LIN {X 0,Y 502.137,Z 842.26,A -85,B 0,C 180,E1 13995.84,E2 13995.84} C_VEL
LIN {X 0,Y 481.443,Z 805.869,A -85,B 0,C 180,E1 13999.134,E2 13999.134} C_VEL
LIN {X 0,Y 469.956,Z 788.258,A -85,B 0,C 180,E1 14001.102,E2 14001.102} C_VEL
LIN {X 0,Y 468.202,Z 783.31,A -85,B 0,C 180,E1 14001.543,E2 14001.543} C_VEL
LIN {X 0,Y 468.344,Z 783.31,A -85,B 0,C 180,E1 14007.257,E2 14007.257} C_VEL
LIN {X 0,Y 468.598,Z 783.31,A -85,B 0,C 180,E1 14013.095,E2 14013.095} C_VEL
LIN {X 0,Y 468.809,Z 783.31,A -85,B 0,C 180,E1 14019.592,E2 14019.592} C_VEL
LIN {X 0,Y 468.958,Z 783.31,A -85,B 0,C 180,E1 14025.753,E2 14025.753} C_VEL
LIN {X 0,Y 469.248,Z 783.31,A -85,B 0,C 180,E1 14030.717,E2 14030.717} C_VEL
LIN {X 0,Y 469.562,Z 783.31,A -85,B 0,C 180,E1 14036.307,E2 14036.307} C_VEL
LIN {X 0,Y 469.678,Z 783.31,A -85,B 0,C 180,E1 14041.855,E2 14041.855} C_VEL
LIN {X 0,Y 469.329,Z 783.31,A -85,B 0,C 180,E1 14047.426,E2 14047.426} C_VEL
LIN {X 0,Y 469.059,Z 783.31,A -85,B 0,C 180,E1 14053.074,E2 14053.074} C_VEL
LIN {X 0,Y 468.787,Z 783.31,A -85,B 0,C 180,E1 14058.863,E2 14058.863} C_VEL
LIN {X 0,Y 468.495,Z 783.31,A -85,B 0,C 180,E1 14065.107,E2 14065.107} C_VEL
LIN {X 0,Y 468.32,Z 783.31,A -85,B 0,C 180,E1 14071.18,E2 14071.18} C_VEL
LIN {X 0,Y 468.157,Z 783.31,A -85,B 0,C 180,E1 14077.951,E2 14077.951} C_VEL
LIN {X 0,Y 468.177,Z 783.696,A -85,B 0,C 180,E1 14081.783,E2 14081.783} C_VEL
LIN {X 0,Y 470.703,Z 789.093,A -85,B 0,C 180,E1 14082.265,E2 14082.265} C_VEL
LIN {X 0,Y 493.353,Z 825.509,A -85,B 0,C 180,E1 14085.963,E2 14085.963} C_VEL
LIN {X 0,Y 512.919,Z 863.779,A -85,B 0,C 180,E1 14089.04,E2 14089.04} C_VEL
LIN {X 0,Y 517.833,Z 877.244,A -85,B 0,C 180,E1 14089.994,E2 14089.994} C_VEL
LIN {X 0,Y 512.74,Z 919.111,A -85,B 0,C 180,E1 14091.466,E2 14091.466} C_VEL
LIN {X 0,Y 506.507,Z 957.08,A -85,B 0,C 180,E1 14093.46,E2 14093.46} C_VEL
LIN {X 0,Y 499.069,Z 993.486,A -85,B 0,C 180,E1 14096.094,E2 14096.094} C_VEL
LIN {X 0,Y 490.992,Z 1028.436,A -85,B 0,C 180,E1 14099.537,E2 14099.537} C_VEL
LIN {X 0,Y 483.283,Z 1059.873,A -85,B 0,C 180,E1 14103.731,E2 14103.731} C_VEL
LIN {X 0,Y 477.35,Z 1085.407,A -85,B 0,C 180,E1 14108.348,E2 14108.348} C_VEL
LIN {X 0,Y 473.318,Z 1105.246,A -85,B 0,C 180,E1 14113.257,E2 14113.257} C_VEL
LIN {X 0,Y 471.002,Z 1119.649,A -85,B 0,C 180,E1 14118.403,E2 14118.403} C_VEL
LIN {X 0,Y 470.112,Z 1128.462,A -85,B 0,C 180,E1 14123.525,E2 14123.525} C_VEL
LIN {X 0,Y 469.91,Z 1132.17,A -85,B 0,C 180,E1 14128.344,E2 14128.344} C_VEL
LIN {X 0,Y 469.969,Z 1131.123,A -85,B 0,C 180,E1 14133.699,E2 14133.699} C_VEL
LIN {X 0,Y 470.403,Z 1125.694,A -85,B 0,C 180,E1 14138.336,E2 14138.336} C_VEL
LIN {X 0,Y 471.702,Z 1114.802,A -85,B 0,C 180,E1 14143.468,E2 14143.468} C_VEL
LIN {X 0,Y 474.604,Z 1098.044,A -85,B 0,C 180,E1 14148.619,E2 14148.619} C_VEL
LIN {X 0,Y 479.46,Z 1075.81,A -85,B 0,C 180,E1 14153.465,E2 14153.465} C_VEL
LIN {X 0,Y 486.177,Z 1048.272,A -85,B 0,C 180,E1 14157.872,E2 14157.872} C_VEL
LIN {X 0,Y 493.802,Z 1016.531,A -85,B 0,C 180,E1 14161.662,E2 14161.662} C_VEL
LIN {X 0,Y 502.224,Z 978.76,A -85,B 0,C 180,E1 14164.976,E2 14164.976} C_VEL
LIN {X 0,Y 509.443,Z 940.342,A -85,B 0,C 180,E1 14167.412,E2 14167.412} C_VEL
LIN {X 0,Y 515.66,Z 896.96,A -85,B 0,C 180,E1 14169.309,E2 14169.309} C_VEL
LIN {X 0,Y 517.573,Z 874.805,A -85,B 0,C 180,E1 14170.015,E2 14170.015} C_VEL
LIN {X 0,Y 499.743,Z 836.77,A -85,B 0,C 180,E1 14172.967,E2 14172.967} C_VEL
LIN {X 0,Y 477.929,Z 800.29,A -85,B 0,C 180,E1 14176.384,E2 14176.384} C_VEL
LIN {X 0,Y 468.27,Z 784.748,A -85,B 0,C 180,E1 14178.066,E2 14178.066} C_VEL
LIN {X 0,Y 468.127,Z 783.31,A -85,B 0,C 180,E1 14178.331,E2 14178.331} C_VEL
LIN {X 0,Y 468.144,Z 783.31,A -85,B 0,C 180,E1 14184.363,E2 14184.363} C_VEL
LIN {X 0,Y 468.406,Z 783.31,A -85,B 0,C 180,E1 14190.856,E2 14190.856} C_VEL
LIN {X 0,Y 468.695,Z 783.31,A -85,B 0,C 180,E1 14197.169,E2 14197.169} C_VEL
LIN {X 0,Y 468.892,Z 783.31,A -85,B 0,C 180,E1 14203.087,E2 14203.087} C_VEL
LIN {X 0,Y 469.159,Z 783.31,A -85,B 0,C 180,E1 14208.821,E2 14208.821} C_VEL
LIN {X 0,Y 469.481,Z 783.31,A -85,B 0,C 180,E1 14214.438,E2 14214.438} C_VEL
LIN {X 0,Y 469.716,Z 783.31,A -85,B 0,C 180,E1 14220.197,E2 14220.197} C_VEL
LIN {X 0,Y 469.484,Z 783.31,A -85,B 0,C 180,E1 14225.549,E2 14225.549} C_VEL
LIN {X 0,Y 469.164,Z 783.31,A -85,B 0,C 180,E1 14231.165,E2 14231.165} C_VEL
LIN {X 0,Y 468.934,Z 783.31,A -85,B 0,C 180,E1 14236.897,E2 14236.897} C_VEL
LIN {X 0,Y 468.69,Z 783.31,A -85,B 0,C 180,E1 14242.816,E2 14242.816} C_VEL
LIN {X 0,Y 468.44,Z 783.31,A -85,B 0,C 180,E1 14249.151,E2 14249.151} C_VEL
LIN {X 0,Y 468.192,Z 783.31,A -85,B 0,C 180,E1 14255.615,E2 14255.615} C_VEL
LIN {X 0,Y 468.162,Z 783.31,A -85,B 0,C 180,E1 14258.52,E2 14258.52} C_VEL
LIN {X 0,Y 470.442,Z 788.792,A -85,B 0,C 180,E1 14259.003,E2 14259.003} C_VEL
LIN {X 0,Y 491.847,Z 823.395,A -85,B 0,C 180,E1 14262.562,E2 14262.562} C_VEL
LIN {X 0,Y 511.25,Z 861.791,A -85,B 0,C 180,E1 14265.703,E2 14265.703} C_VEL
LIN {X 0,Y 517.752,Z 880.2,A -85,B 0,C 180,E1 14267.006,E2 14267.006} C_VEL
LIN {X 0,Y 511.952,Z 925.172,A -85,B 0,C 180,E1 14268.671,E2 14268.671} C_VEL
LIN {X 0,Y 505.377,Z 965.131,A -85,B 0,C 180,E1 14270.845,E2 14270.845} C_VEL
LIN {X 0,Y 497.792,Z 1003.837,A -85,B 0,C 180,E1 14273.696,E2 14273.696} C_VEL
LIN {X 0,Y 490.044,Z 1040.04,A -85,B 0,C 180,E1 14277.241,E2 14277.241} C_VEL
LIN {X 0,Y 482.582,Z 1073.759,A -85,B 0,C 180,E1 14281.611,E2 14281.611} C_VEL
LIN {X 0,Y 476.669,Z 1102.525,A -85,B 0,C 180,E1 14286.581,E2 14286.581} C_VEL
LIN {X 0,Y 472.768,Z 1124.824,A -85,B 0,C 180,E1 14291.79,E2 14291.79} C_VEL
LIN {X 0,Y 470.811,Z 1140.724,A -85,B 0,C 180,E1 14296.979,E2 14296.979} C_VEL
LIN {X 0,Y 470.084,Z 1150.402,A -85,B 0,C 180,E1 14301.659,E2 14301.659} C_VEL
LIN {X 0,Y 469.852,Z 1155.82,A -85,B 0,C 180,E1 14306.452,E2 14306.452} C_VEL
LIN {X 0,Y 469.839,Z 1156.983,A -85,B 0,C 180,E1 14310.59,E2 14310.59} C_VEL
LIN {X 0,Y 467.269,Z 1156.571,A -85,B 0,C 180,E1 14312.158,E2 14312.158} C_VEL
LIN {X 0,Y 462.037,Z 1154.958,A -85,B 0,C 180,E1 14314.507,E2 14314.507} C_VEL
LIN {X 0,Y 461.956,Z 1154.639,A -85,B 0,C 180,E1 14314.778,E2 14314.778} C_VEL
LIN {X 0,Y 462.381,Z 1147.514,A -85,B 0,C 180,E1 14320.05,E2 14320.05} C_VEL
LIN {X 0,Y 463.607,Z 1135.397,A -85,B 0,C 180,E1 14325.155,E2 14325.155} C_VEL
LIN {X 0,Y 466.042,Z 1118.859,A -85,B 0,C 180,E1 14330.06,E2 14330.06} C_VEL
LIN {X 0,Y 470.798,Z 1094.464,A -85,B 0,C 180,E1 14335.333,E2 14335.333} C_VEL
LIN {X 0,Y 477.18,Z 1065.586,A -85,B 0,C 180,E1 14340.005,E2 14340.005} C_VEL
LIN {X 0,Y 484.532,Z 1033.657,A -85,B 0,C 180,E1 14343.954,E2 14343.954} C_VEL
LIN {X 0,Y 492.668,Z 997.08,A -85,B 0,C 180,E1 14347.407,E2 14347.407} C_VEL
LIN {X 0,Y 500.674,Z 956.87,A -85,B 0,C 180,E1 14350.236,E2 14350.236} C_VEL
LIN {X 0,Y 507.726,Z 913.166,A -85,B 0,C 180,E1 14352.431,E2 14352.431} C_VEL
LIN {X 0,Y 511.182,Z 880.089,A -85,B 0,C 180,E1 14353.66,E2 14353.66} C_VEL
LIN {X 0,Y 495.285,Z 843.197,A -85,B 0,C 180,E1 14356.593,E2 14356.593} C_VEL
LIN {X 0,Y 474.161,Z 806.529,A -85,B 0,C 180,E1 14360.088,E2 14360.088} C_VEL
LIN {X 0,Y 462.098,Z 788.373,A -85,B 0,C 180,E1 14362.252,E2 14362.252} C_VEL
LIN {X 0,Y 460.222,Z 783.31,A -85,B 0,C 180,E1 14362.767,E2 14362.767} C_VEL
LIN {X 0,Y 460.431,Z 783.31,A -85,B 0,C 180,E1 14368.822,E2 14368.822} C_VEL
LIN {X 0,Y 460.701,Z 783.31,A -85,B 0,C 180,E1 14374.698,E2 14374.698} C_VEL
LIN {X 0,Y 460.903,Z 783.31,A -85,B 0,C 180,E1 14380.817,E2 14380.817} C_VEL
LIN {X 0,Y 461.081,Z 783.31,A -85,B 0,C 180,E1 14386.71,E2 14386.71} C_VEL
LIN {X 0,Y 461.405,Z 783.31,A -85,B 0,C 180,E1 14392.46,E2 14392.46} C_VEL
LIN {X 0,Y 461.694,Z 783.31,A -85,B 0,C 180,E1 14398.127,E2 14398.127} C_VEL
LIN {X 0,Y 461.638,Z 783.31,A -85,B 0,C 180,E1 14403.77,E2 14403.77} C_VEL
LIN {X 0,Y 461.265,Z 783.31,A -85,B 0,C 180,E1 14409.8,E2 14409.8} C_VEL
LIN {X 0,Y 461.045,Z 783.31,A -85,B 0,C 180,E1 14415.249,E2 14415.249} C_VEL
LIN {X 0,Y 460.771,Z 783.31,A -85,B 0,C 180,E1 14421.211,E2 14421.211} C_VEL
LIN {X 0,Y 460.494,Z 783.31,A -85,B 0,C 180,E1 14427.434,E2 14427.434} C_VEL
LIN {X 0,Y 460.404,Z 783.31,A -85,B 0,C 180,E1 14431.778,E2 14431.778} C_VEL
LIN {X 0,Y 460.242,Z 783.31,A -85,B 0,C 180,E1 14438.724,E2 14438.724} C_VEL
LIN {X 0,Y 460.28,Z 784.013,A -85,B 0,C 180,E1 14440.607,E2 14440.607} C_VEL
LIN {X 0,Y 463.069,Z 789.376,A -85,B 0,C 180,E1 14441.157,E2 14441.157} C_VEL
LIN {X 0,Y 485.801,Z 825.573,A -85,B 0,C 180,E1 14445.044,E2 14445.044} C_VEL
LIN {X 0,Y 505.461,Z 863.424,A -85,B 0,C 180,E1 14448.247,E2 14448.247} C_VEL
LIN {X 0,Y 511.686,Z 879.986,A -85,B 0,C 180,E1 14449.476,E2 14449.476} C_VEL
LIN {X 0,Y 505.894,Z 924.716,A -85,B 0,C 180,E1 14451.131,E2 14451.131} C_VEL
LIN {X 0,Y 498.37,Z 966.506,A -85,B 0,C 180,E1 14453.491,E2 14453.491} C_VEL
LIN {X 0,Y 489.997,Z 1004.78,A -85,B 0,C 180,E1 14456.556,E2 14456.556} C_VEL
LIN {X 0,Y 481.625,Z 1038.934,A -85,B 0,C 180,E1 14460.3,E2 14460.3} C_VEL
LIN {X 0,Y 474.021,Z 1068.554,A -85,B 0,C 180,E1 14464.692,E2 14464.692} C_VEL
LIN {X 0,Y 468.197,Z 1092.887,A -85,B 0,C 180,E1 14469.62,E2 14469.62} C_VEL
LIN {X 0,Y 464.543,Z 1111.412,A -85,B 0,C 180,E1 14474.876,E2 14474.876} C_VEL
LIN {X 0,Y 462.804,Z 1123.156,A -85,B 0,C 180,E1 14479.827,E2 14479.827} C_VEL
LIN {X 0,Y 462.149,Z 1129.779,A -85,B 0,C 180,E1 14484.357,E2 14484.357} C_VEL
LIN {X 0,Y 462.116,Z 1132.652,A -85,B 0,C 180,E1 14490.002,E2 14490.002} C_VEL
LIN {X 0,Y 462.161,Z 1129.692,A -85,B 0,C 180,E1 14495.646,E2 14495.646} C_VEL
LIN {X 0,Y 463.026,Z 1121.405,A -85,B 0,C 180,E1 14500.971,E2 14500.971} C_VEL
LIN {X 0,Y 465.206,Z 1107.528,A -85,B 0,C 180,E1 14506.28,E2 14506.28} C_VEL
LIN {X 0,Y 469.239,Z 1088.397,A -85,B 0,C 180,E1 14511.302,E2 14511.302} C_VEL
LIN {X 0,Y 474.841,Z 1065.186,A -85,B 0,C 180,E1 14515.772,E2 14515.772} C_VEL
LIN {X 0,Y 482.135,Z 1036.352,A -85,B 0,C 180,E1 14519.928,E2 14519.928} C_VEL
LIN {X 0,Y 490.088,Z 1004.144,A -85,B 0,C 180,E1 14523.408,E2 14523.408} C_VEL
LIN {X 0,Y 498.525,Z 965.577,A -85,B 0,C 180,E1 14526.471,E2 14526.471} C_VEL
LIN {X 0,Y 506.007,Z 923.833,A -85,B 0,C 180,E1 14528.807,E2 14528.807} C_VEL
LIN {X 0,Y 511.644,Z 880.67,A -85,B 0,C 180,E1 14530.401,E2 14530.401} C_VEL
LIN {X 0,Y 510.204,Z 874.376,A -85,B 0,C 180,E1 14530.773,E2 14530.773} C_VEL
LIN {X 0,Y 492.269,Z 836.832,A -85,B 0,C 180,E1 14533.832,E2 14533.832} C_VEL
LIN {X 0,Y 470.597,Z 800.932,A -85,B 0,C 180,E1 14537.375,E2 14537.375} C_VEL
LIN {X 0,Y 461.857,Z 788.163,A -85,B 0,C 180,E1 14538.936,E2 14538.936} C_VEL
LIN {X 0,Y 460.231,Z 783.31,A -85,B 0,C 180,E1 14539.376,E2 14539.376} C_VEL
LIN {X 0,Y 460.254,Z 783.31,A -85,B 0,C 180,E1 14545.964,E2 14545.964} C_VEL
LIN {X 0,Y 460.453,Z 783.31,A -85,B 0,C 180,E1 14550.418,E2 14550.418} C_VEL
LIN {X 0,Y 460.768,Z 783.31,A -85,B 0,C 180,E1 14557.038,E2 14557.038} C_VEL
LIN {X 0,Y 460.943,Z 783.31,A -85,B 0,C 180,E1 14562.786,E2 14562.786} C_VEL
LIN {X 0,Y 461.221,Z 783.31,A -85,B 0,C 180,E1 14568.626,E2 14568.626} C_VEL
LIN {X 0,Y 461.563,Z 783.31,A -85,B 0,C 180,E1 14574.342,E2 14574.342} C_VEL
LIN {X 0,Y 461.888,Z 783.31,A -85,B 0,C 180,E1 14579.993,E2 14579.993} C_VEL
LIN {X 0,Y 461.563,Z 783.31,A -85,B 0,C 180,E1 14585.644,E2 14585.644} C_VEL
LIN {X 0,Y 461.26,Z 783.31,A -85,B 0,C 180,E1 14591.359,E2 14591.359} C_VEL
LIN {X 0,Y 460.946,Z 783.31,A -85,B 0,C 180,E1 14597.584,E2 14597.584} C_VEL
LIN {X 0,Y 460.736,Z 783.31,A -85,B 0,C 180,E1 14603.233,E2 14603.233} C_VEL
LIN {X 0,Y 460.487,Z 783.31,A -85,B 0,C 180,E1 14609.563,E2 14609.563} C_VEL
LIN {X 0,Y 460.261,Z 783.31,A -85,B 0,C 180,E1 14616.326,E2 14616.326} C_VEL
LIN {X 0,Y 460.219,Z 783.31,A -85,B 0,C 180,E1 14617.355,E2 14617.355} C_VEL
LIN {X 0,Y 462.411,Z 788.688,A -85,B 0,C 180,E1 14617.83,E2 14617.83} C_VEL
LIN {X 0,Y 481.73,Z 818.938,A -85,B 0,C 180,E1 14621.215,E2 14621.215} C_VEL
LIN {X 0,Y 501.601,Z 856.645,A -85,B 0,C 180,E1 14624.522,E2 14624.522} C_VEL
LIN {X 0,Y 511.607,Z 881.901,A -85,B 0,C 180,E1 14626.472,E2 14626.472} C_VEL
LIN {X 0,Y 505.544,Z 927.284,A -85,B 0,C 180,E1 14628.19,E2 14628.19} C_VEL
LIN {X 0,Y 498.093,Z 970.128,A -85,B 0,C 180,E1 14630.607,E2 14630.607} C_VEL
LIN {X 0,Y 489.954,Z 1009.59,A -85,B 0,C 180,E1 14633.677,E2 14633.677} C_VEL
LIN {X 0,Y 482.234,Z 1043.786,A -85,B 0,C 180,E1 14637.199,E2 14637.199} C_VEL
LIN {X 0,Y 474.966,Z 1075.184,A -85,B 0,C 180,E1 14641.41,E2 14641.41} C_VEL
LIN {X 0,Y 469.162,Z 1102.286,A -85,B 0,C 180,E1 14646.189,E2 14646.189} C_VEL
LIN {X 0,Y 465.032,Z 1124.579,A -85,B 0,C 180,E1 14651.476,E2 14651.476} C_VEL
LIN {X 0,Y 462.975,Z 1140.496,A -85,B 0,C 180,E1 14656.755,E2 14656.755} C_VEL
LIN {X 0,Y 462.195,Z 1150.185,A -85,B 0,C 180,E1 14661.515,E2 14661.515} C_VEL
LIN {X 0,Y 461.969,Z 1155.529,A -85,B 0,C 180,E1 14666.237,E2 14666.237} C_VEL
LIN {X 0,Y 461.952,Z 1156.781,A -85,B 0,C 180,E1 14670.578,E2 14670.578} C_VEL
LIN {X 0,Y 461.956,Z 1154.639,A -85,B 0,C 180,E1 14674.778,E2 14674.778} C_VEL
LIN {X 0,Y 459.513,Z 1153.086,A -85,B 0,C 180,E1 14676.37,E2 14676.37} C_VEL
LIN {X 0,Y 454.377,Z 1149.794,A -85,B 0,C 180,E1 14678.746,E2 14678.746} C_VEL
LIN {X 0,Y 454.313,Z 1149.329,A -85,B 0,C 180,E1 14679.018,E2 14679.018} C_VEL
LIN {X 0,Y 455.438,Z 1137.912,A -85,B 0,C 180,E1 14684.447,E2 14684.447} C_VEL
LIN {X 0,Y 458.108,Z 1120.133,A -85,B 0,C 180,E1 14689.998,E2 14689.998} C_VEL
LIN {X 0,Y 462.719,Z 1097.128,A -85,B 0,C 180,E1 14695.192,E2 14695.192} C_VEL
LIN {X 0,Y 468.982,Z 1070.216,A -85,B 0,C 180,E1 14699.782,E2 14699.782} C_VEL
LIN {X 0,Y 476.827,Z 1037.265,A -85,B 0,C 180,E1 14704.074,E2 14704.074} C_VEL
LIN {X 0,Y 485.758,Z 998.947,A -85,B 0,C 180,E1 14707.807,E2 14707.807} C_VEL
LIN {X 0,Y 494.299,Z 957.741,A -85,B 0,C 180,E1 14710.76,E2 14710.76} C_VEL
LIN {X 0,Y 501.416,Z 915.123,A -85,B 0,C 180,E1 14712.939,E2 14712.939} C_VEL
LIN {X 0,Y 504.969,Z 882.722,A -85,B 0,C 180,E1 14714.182,E2 14714.182} C_VEL
LIN {X 0,Y 489.322,Z 845.888,A -85,B 0,C 180,E1 14717.226,E2 14717.226} C_VEL
LIN {X 0,Y 468.955,Z 810.661,A -85,B 0,C 180,E1 14720.712,E2 14720.712} C_VEL
LIN {X 0,Y 454.386,Z 788.622,A -85,B 0,C 180,E1 14723.443,E2 14723.443} C_VEL
LIN {X 0,Y 452.347,Z 783.31,A -85,B 0,C 180,E1 14723.989,E2 14723.989} C_VEL
LIN {X 0,Y 452.593,Z 783.31,A -85,B 0,C 180,E1 14730.503,E2 14730.503} C_VEL
LIN {X 0,Y 452.793,Z 783.31,A -85,B 0,C 180,E1 14736.335,E2 14736.335} C_VEL
LIN {X 0,Y 453.029,Z 783.31,A -85,B 0,C 180,E1 14742.491,E2 14742.491} C_VEL
LIN {X 0,Y 453.273,Z 783.31,A -85,B 0,C 180,E1 14748.439,E2 14748.439} C_VEL
LIN {X 0,Y 453.644,Z 783.31,A -85,B 0,C 180,E1 14754.257,E2 14754.257} C_VEL
LIN {X 0,Y 453.945,Z 783.31,A -85,B 0,C 180,E1 14760.007,E2 14760.007} C_VEL
LIN {X 0,Y 453.669,Z 783.31,A -85,B 0,C 180,E1 14765.757,E2 14765.757} C_VEL
LIN {X 0,Y 453.31,Z 783.31,A -85,B 0,C 180,E1 14771.575,E2 14771.575} C_VEL
LIN {X 0,Y 452.998,Z 783.31,A -85,B 0,C 180,E1 14777.525,E2 14777.525} C_VEL
LIN {X 0,Y 452.703,Z 783.31,A -85,B 0,C 180,E1 14783.686,E2 14783.686} C_VEL
LIN {X 0,Y 452.523,Z 783.31,A -85,B 0,C 180,E1 14790.153,E2 14790.153} C_VEL
LIN {X 0,Y 452.336,Z 783.31,A -85,B 0,C 180,E1 14797.085,E2 14797.085} C_VEL
LIN {X 0,Y 452.362,Z 783.985,A -85,B 0,C 180,E1 14799.351,E2 14799.351} C_VEL
LIN {X 0,Y 455.094,Z 789.271,A -85,B 0,C 180,E1 14799.92,E2 14799.92} C_VEL
LIN {X 0,Y 477.815,Z 824.741,A -85,B 0,C 180,E1 14804.004,E2 14804.004} C_VEL
LIN {X 0,Y 497.179,Z 861.253,A -85,B 0,C 180,E1 14807.272,E2 14807.272} C_VEL
LIN {X 0,Y 505.597,Z 882.275,A -85,B 0,C 180,E1 14808.939,E2 14808.939} C_VEL
LIN {X 0,Y 499.674,Z 925.842,A -85,B 0,C 180,E1 14810.591,E2 14810.591} C_VEL
LIN {X 0,Y 491.813,Z 967.814,A -85,B 0,C 180,E1 14813.006,E2 14813.006} C_VEL
LIN {X 0,Y 483.36,Z 1005.141,A -85,B 0,C 180,E1 14816.039,E2 14816.039} C_VEL
LIN {X 0,Y 474.65,Z 1039.217,A -85,B 0,C 180,E1 14819.819,E2 14819.819} C_VEL
LIN {X 0,Y 466.765,Z 1068.809,A -85,B 0,C 180,E1 14824.27,E2 14824.27} C_VEL
LIN {X 0,Y 460.663,Z 1093.122,A -85,B 0,C 180,E1 14829.271,E2 14829.271} C_VEL
LIN {X 0,Y 456.803,Z 1111.635,A -85,B 0,C 180,E1 14834.614,E2 14834.614} C_VEL
LIN {X 0,Y 454.948,Z 1123.591,A -85,B 0,C 180,E1 14839.763,E2 14839.763} C_VEL
LIN {X 0,Y 454.275,Z 1129.988,A -85,B 0,C 180,E1 14844.259,E2 14844.259} C_VEL
LIN {X 0,Y 454.223,Z 1132.859,A -85,B 0,C 180,E1 14850.002,E2 14850.002} C_VEL
LIN {X 0,Y 454.287,Z 1129.901,A -85,B 0,C 180,E1 14855.744,E2 14855.744} C_VEL
LIN {X 0,Y 455.128,Z 1122.057,A -85,B 0,C 180,E1 14860.937,E2 14860.937} C_VEL
LIN {X 0,Y 457.169,Z 1109.423,A -85,B 0,C 180,E1 14866.021,E2 14866.021} C_VEL
LIN {X 0,Y 461.252,Z 1090.757,A -85,B 0,C 180,E1 14871.184,E2 14871.184} C_VEL
LIN {X 0,Y 467.256,Z 1066.882,A -85,B 0,C 180,E1 14875.963,E2 14875.963} C_VEL
LIN {X 0,Y 475.072,Z 1037.165,A -85,B 0,C 180,E1 14880.348,E2 14880.348} C_VEL
LIN {X 0,Y 483.785,Z 1003.021,A -85,B 0,C 180,E1 14884.062,E2 14884.062} C_VEL
LIN {X 0,Y 492.194,Z 965.883,A -85,B 0,C 180,E1 14887.029,E2 14887.029} C_VEL
LIN {X 0,Y 499.901,Z 924.442,A -85,B 0,C 180,E1 14889.372,E2 14889.372} C_VEL
LIN {X 0,Y 505.388,Z 880.472,A -85,B 0,C 180,E1 14891.052,E2 14891.052} C_VEL
LIN {X 0,Y 487.948,Z 842.58,A -85,B 0,C 180,E1 14894.214,E2 14894.214} C_VEL
LIN {X 0,Y 466.405,Z 806.497,A -85,B 0,C 180,E1 14897.848,E2 14897.848} C_VEL
LIN {X 0,Y 454.269,Z 788.526,A -85,B 0,C 180,E1 14900.11,E2 14900.11} C_VEL
LIN {X 0,Y 452.293,Z 783.31,A -85,B 0,C 180,E1 14900.706,E2 14900.706} C_VEL
LIN {X 0,Y 452.381,Z 783.31,A -85,B 0,C 180,E1 14907.591,E2 14907.591} C_VEL
LIN {X 0,Y 452.546,Z 783.31,A -85,B 0,C 180,E1 14912.043,E2 14912.043} C_VEL
LIN {X 0,Y 452.872,Z 783.31,A -85,B 0,C 180,E1 14918.401,E2 14918.401} C_VEL
LIN {X 0,Y 453.083,Z 783.31,A -85,B 0,C 180,E1 14924.477,E2 14924.477} C_VEL
LIN {X 0,Y 453.448,Z 783.31,A -85,B 0,C 180,E1 14930.376,E2 14930.376} C_VEL
LIN {X 0,Y 453.753,Z 783.31,A -85,B 0,C 180,E1 14936.164,E2 14936.164} C_VEL
LIN {X 0,Y 453.894,Z 783.31,A -85,B 0,C 180,E1 14941.906,E2 14941.906} C_VEL
LIN {X 0,Y 453.507,Z 783.31,A -85,B 0,C 180,E1 14947.672,E2 14947.672} C_VEL
LIN {X 0,Y 453.164,Z 783.31,A -85,B 0,C 180,E1 14954.153,E2 14954.153} C_VEL
LIN {X 0,Y 452.883,Z 783.31,A -85,B 0,C 180,E1 14960.48,E2 14960.48} C_VEL
LIN {X 0,Y 452.691,Z 783.31,A -85,B 0,C 180,E1 14965.782,E2 14965.782} C_VEL
LIN {X 0,Y 452.414,Z 783.31,A -85,B 0,C 180,E1 14972.39,E2 14972.39} C_VEL
LIN {X 0,Y 452.384,Z 784.025,A -85,B 0,C 180,E1 14976.142,E2 14976.142} C_VEL
LIN {X 0,Y 455.133,Z 789.322,A -85,B 0,C 180,E1 14976.722,E2 14976.722} C_VEL
LIN {X 0,Y 476.66,Z 823.182,A -85,B 0,C 180,E1 14980.651,E2 14980.651} C_VEL
LIN {X 0,Y 495.972,Z 860.36,A -85,B 0,C 180,E1 14984.013,E2 14984.013} C_VEL
LIN {X 0,Y 505.355,Z 884.785,A -85,B 0,C 180,E1 14985.963,E2 14985.963} C_VEL
LIN {X 0,Y 499.243,Z 928.689,A -85,B 0,C 180,E1 14987.67,E2 14987.67} C_VEL
LIN {X 0,Y 491.498,Z 971.707,A -85,B 0,C 180,E1 14990.142,E2 14990.142} C_VEL
LIN {X 0,Y 482.747,Z 1012.382,A -85,B 0,C 180,E1 14993.39,E2 14993.39} C_VEL
LIN {X 0,Y 474.239,Z 1048.3,A -85,B 0,C 180,E1 14997.247,E2 14997.247} C_VEL
LIN {X 0,Y 466.637,Z 1079.535,A -85,B 0,C 180,E1 15001.673,E2 15001.673} C_VEL
LIN {X 0,Y 461.017,Z 1105.412,A -85,B 0,C 180,E1 15006.514,E2 15006.514} C_VEL
LIN {X 0,Y 457.088,Z 1126.08,A -85,B 0,C 180,E1 15011.643,E2 15011.643} C_VEL
LIN {X 0,Y 455.035,Z 1141.459,A -85,B 0,C 180,E1 15017.01,E2 15017.01} C_VEL
LIN {X 0,Y 454.317,Z 1149.969,A -85,B 0,C 180,E1 15021.367,E2 15021.367} C_VEL
LIN {X 0,Y 454.065,Z 1155.32,A -85,B 0,C 180,E1 15026.172,E2 15026.172} C_VEL
LIN {X 0,Y 454.165,Z 1156.682,A -85,B 0,C 180,E1 15029.998,E2 15029.998} C_VEL
LIN {X 0,Y 454.164,Z 1153.668,A -85,B 0,C 180,E1 15035.742,E2 15035.742} C_VEL
LIN {X 0,Y 454.313,Z 1149.329,A -85,B 0,C 180,E1 15039.018,E2 15039.018} C_VEL
LIN {X 0,Y 453.2,Z 1147.54,A -85,B 0,C 180,E1 15040.09,E2 15040.09} C_VEL
LIN {X 0,Y 447.22,Z 1141.789,A -85,B 0,C 180,E1 15042.998,E2 15042.998} C_VEL
LIN {X 0,Y 447.198,Z 1141.136,A -85,B 0,C 180,E1 15043.269,E2 15043.269} C_VEL
LIN {X 0,Y 449.348,Z 1126.179,A -85,B 0,C 180,E1 15048.583,E2 15048.583} C_VEL
LIN {X 0,Y 453.715,Z 1104.081,A -85,B 0,C 180,E1 15054.145,E2 15054.145} C_VEL
LIN {X 0,Y 459.678,Z 1078.542,A -85,B 0,C 180,E1 15058.933,E2 15058.933} C_VEL
LIN {X 0,Y 467.261,Z 1048.542,A -85,B 0,C 180,E1 15063.237,E2 15063.237} C_VEL
LIN {X 0,Y 476.204,Z 1012.16,A -85,B 0,C 180,E1 15067.193,E2 15067.193} C_VEL
LIN {X 0,Y 485.224,Z 972.136,A -85,B 0,C 180,E1 15070.416,E2 15070.416} C_VEL
LIN {X 0,Y 493.15,Z 929.329,A -85,B 0,C 180,E1 15072.909,E2 15072.909} C_VEL
LIN {X 0,Y 498.869,Z 885.478,A -85,B 0,C 180,E1 15074.702,E2 15074.702} C_VEL
LIN {X 0,Y 483.897,Z 849.707,A -85,B 0,C 180,E1 15077.775,E2 15077.775} C_VEL
LIN {X 0,Y 463.201,Z 813.384,A -85,B 0,C 180,E1 15081.474,E2 15081.474} C_VEL
LIN {X 0,Y 446.905,Z 789.046,A -85,B 0,C 180,E1 15084.669,E2 15084.669} C_VEL
LIN {X 0,Y 444.556,Z 784.565,A -85,B 0,C 180,E1 15085.196,E2 15085.196} C_VEL
LIN {X 0,Y 444.469,Z 783.31,A -85,B 0,C 180,E1 15085.4,E2 15085.4} C_VEL
LIN {X 0,Y 444.731,Z 783.31,A -85,B 0,C 180,E1 15092.346,E2 15092.346} C_VEL
LIN {X 0,Y 444.907,Z 783.31,A -85,B 0,C 180,E1 15098.01,E2 15098.01} C_VEL
LIN {X 0,Y 445.135,Z 783.31,A -85,B 0,C 180,E1 15104.208,E2 15104.208} C_VEL
LIN {X 0,Y 445.5,Z 783.31,A -85,B 0,C 180,E1 15110.494,E2 15110.494} C_VEL
LIN {X 0,Y 445.828,Z 783.31,A -85,B 0,C 180,E1 15116.11,E2 15116.11} C_VEL
LIN {X 0,Y 445.963,Z 783.31,A -85,B 0,C 180,E1 15121.954,E2 15121.954} C_VEL
LIN {X 0,Y 445.571,Z 783.31,A -85,B 0,C 180,E1 15127.824,E2 15127.824} C_VEL
LIN {X 0,Y 445.272,Z 783.31,A -85,B 0,C 180,E1 15133.786,E2 15133.786} C_VEL
LIN {X 0,Y 444.973,Z 783.31,A -85,B 0,C 180,E1 15139.914,E2 15139.914} C_VEL
LIN {X 0,Y 444.633,Z 783.31,A -85,B 0,C 180,E1 15146.301,E2 15146.301} C_VEL
LIN {X 0,Y 444.474,Z 783.31,A -85,B 0,C 180,E1 15153.059,E2 15153.059} C_VEL
LIN {X 0,Y 444.418,Z 783.31,A -85,B 0,C 180,E1 15157.969,E2 15157.969} C_VEL
LIN {X 0,Y 446.657,Z 788.781,A -85,B 0,C 180,E1 15158.515,E2 15158.515} C_VEL
LIN {X 0,Y 463.732,Z 814.14,A -85,B 0,C 180,E1 15161.82,E2 15161.82} C_VEL
LIN {X 0,Y 484.834,Z 850.729,A -85,B 0,C 180,E1 15165.492,E2 15165.492} C_VEL
LIN {X 0,Y 499.523,Z 884.764,A -85,B 0,C 180,E1 15168.405,E2 15168.405} C_VEL
LIN {X 0,Y 493.485,Z 927.025,A -85,B 0,C 180,E1 15170.043,E2 15170.043} C_VEL
LIN {X 0,Y 485.625,Z 967.801,A -85,B 0,C 180,E1 15172.416,E2 15172.416} C_VEL
LIN {X 0,Y 476.941,Z 1004.895,A -85,B 0,C 180,E1 15175.449,E2 15175.449} C_VEL
LIN {X 0,Y 467.825,Z 1039.078,A -85,B 0,C 180,E1 15179.266,E2 15179.266} C_VEL
LIN {X 0,Y 459.511,Z 1069.062,A -85,B 0,C 180,E1 15183.833,E2 15183.833} C_VEL
LIN {X 0,Y 453.237,Z 1092.941,A -85,B 0,C 180,E1 15188.803,E2 15188.803} C_VEL
LIN {X 0,Y 449.061,Z 1111.857,A -85,B 0,C 180,E1 15194.342,E2 15194.342} C_VEL
LIN {X 0,Y 447.129,Z 1123.352,A -85,B 0,C 180,E1 15199.341,E2 15199.341} C_VEL
LIN {X 0,Y 446.385,Z 1130.197,A -85,B 0,C 180,E1 15204.157,E2 15204.157} C_VEL
LIN {X 0,Y 446.324,Z 1133.066,A -85,B 0,C 180,E1 15210.002,E2 15210.002} C_VEL
LIN {X 0,Y 446.399,Z 1130.111,A -85,B 0,C 180,E1 15215.846,E2 15215.846} C_VEL
LIN {X 0,Y 447.201,Z 1123.073,A -85,B 0,C 180,E1 15220.708,E2 15220.708} C_VEL
LIN {X 0,Y 449.111,Z 1111.586,A -85,B 0,C 180,E1 15225.66,E2 15225.66} C_VEL
LIN {X 0,Y 453.41,Z 1092.501,A -85,B 0,C 180,E1 15231.204,E2 15231.204} C_VEL
LIN {X 0,Y 459.668,Z 1068.549,A -85,B 0,C 180,E1 15236.161,E2 15236.161} C_VEL
LIN {X 0,Y 467.914,Z 1038.47,A -85,B 0,C 180,E1 15240.719,E2 15240.719} C_VEL
LIN {X 0,Y 477.189,Z 1003.446,A -85,B 0,C 180,E1 15244.591,E2 15244.591} C_VEL
LIN {X 0,Y 486.052,Z 965.454,A -85,B 0,C 180,E1 15247.65,E2 15247.65} C_VEL
LIN {X 0,Y 493.878,Z 924.84,A -85,B 0,C 180,E1 15249.959,E2 15249.959} C_VEL
LIN {X 0,Y 499.104,Z 882.863,A -85,B 0,C 180,E1 15251.621,E2 15251.621} C_VEL
LIN {X 0,Y 482.61,Z 846.442,A -85,B 0,C 180,E1 15254.778,E2 15254.778} C_VEL
LIN {X 0,Y 461.976,Z 811.64,A -85,B 0,C 180,E1 15258.378,E2 15258.378} C_VEL
LIN {X 0,Y 446.691,Z 788.884,A -85,B 0,C 180,E1 15261.353,E2 15261.353} C_VEL
LIN {X 0,Y 444.385,Z 783.31,A -85,B 0,C 180,E1 15261.928,E2 15261.928} C_VEL
LIN {X 0,Y 444.482,Z 783.31,A -85,B 0,C 180,E1 15268.456,E2 15268.456} C_VEL
LIN {X 0,Y 444.665,Z 783.31,A -85,B 0,C 180,E1 15273.701,E2 15273.701} C_VEL
LIN {X 0,Y 445.017,Z 783.31,A -85,B 0,C 180,E1 15280.088,E2 15280.088} C_VEL
LIN {X 0,Y 445.253,Z 783.31,A -85,B 0,C 180,E1 15286.213,E2 15286.213} C_VEL
LIN {X 0,Y 445.612,Z 783.31,A -85,B 0,C 180,E1 15292.256,E2 15292.256} C_VEL
LIN {X 0,Y 445.933,Z 783.31,A -85,B 0,C 180,E1 15298.046,E2 15298.046} C_VEL
LIN {X 0,Y 445.836,Z 783.31,A -85,B 0,C 180,E1 15303.89,E2 15303.89} C_VEL
LIN {X 0,Y 445.512,Z 783.31,A -85,B 0,C 180,E1 15309.782,E2 15309.782} C_VEL
LIN {X 0,Y 445.207,Z 783.31,A -85,B 0,C 180,E1 15315.79,E2 15315.79} C_VEL
LIN {X 0,Y 444.9,Z 783.31,A -85,B 0,C 180,E1 15321.991,E2 15321.991} C_VEL
LIN {X 0,Y 444.68,Z 783.31,A -85,B 0,C 180,E1 15328.48,E2 15328.48} C_VEL
LIN {X 0,Y 444.486,Z 783.823,A -85,B 0,C 180,E1 15334.807,E2 15334.807} C_VEL
LIN {X 0,Y 447.05,Z 789.176,A -85,B 0,C 180,E1 15335.392,E2 15335.392} C_VEL
LIN {X 0,Y 467.199,Z 820.125,A -85,B 0,C 180,E1 15339.289,E2 15339.289} C_VEL
LIN {X 0,Y 486.571,Z 855.739,A -85,B 0,C 180,E1 15342.77,E2 15342.77} C_VEL
LIN {X 0,Y 499.202,Z 887.297,A -85,B 0,C 180,E1 15345.431,E2 15345.431} C_VEL
LIN {X 0,Y 493.153,Z 929.112,A -85,B 0,C 180,E1 15347.09,E2 15347.09} C_VEL
LIN {X 0,Y 485.21,Z 971.766,A -85,B 0,C 180,E1 15349.563,E2 15349.563} C_VEL
LIN {X 0,Y 476.205,Z 1012.016,A -85,B 0,C 180,E1 15352.803,E2 15352.803} C_VEL
LIN {X 0,Y 467.273,Z 1048.44,A -85,B 0,C 180,E1 15356.76,E2 15356.76} C_VEL
LIN {X 0,Y 459.311,Z 1079.875,A -85,B 0,C 180,E1 15361.291,E2 15361.291} C_VEL
LIN {X 0,Y 453.474,Z 1105.157,A -85,B 0,C 180,E1 15366.099,E2 15366.099} C_VEL
LIN {X 0,Y 449.308,Z 1126.167,A -85,B 0,C 180,E1 15371.417,E2 15371.417} C_VEL
LIN {X 0,Y 447.076,Z 1142.421,A -85,B 0,C 180,E1 15377.272,E2 15377.272} C_VEL
LIN {X 0,Y 446.336,Z 1151.126,A -85,B 0,C 180,E1 15382.194,E2 15382.194} C_VEL
LIN {X 0,Y 446.162,Z 1155.112,A -85,B 0,C 180,E1 15386.104,E2 15386.104} C_VEL
LIN {X 0,Y 446.266,Z 1156.475,A -85,B 0,C 180,E1 15389.998,E2 15389.998} C_VEL
LIN {X 0,Y 446.265,Z 1153.458,A -85,B 0,C 180,E1 15395.844,E2 15395.844} C_VEL
LIN {X 0,Y 446.707,Z 1146.193,A -85,B 0,C 180,E1 15400.88,E2 15400.88} C_VEL
LIN {X 0,Y 447.198,Z 1141.136,A -85,B 0,C 180,E1 15403.269,E2 15403.269} C_VEL
LIN {X 0,Y 444.018,Z 1136.104,A -85,B 0,C 180,E1 15405.389,E2 15405.389} C_VEL
LIN {X 0,Y 440.96,Z 1130.356,A -85,B 0,C 180,E1 15407.509,E2 15407.509} C_VEL
LIN {X 0,Y 444.971,Z 1109.921,A -85,B 0,C 180,E1 15413.196,E2 15413.196} C_VEL
LIN {X 0,Y 451.292,Z 1083.065,A -85,B 0,C 180,E1 15418.64,E2 15418.64} C_VEL
LIN {X 0,Y 459.828,Z 1050.736,A -85,B 0,C 180,E1 15423.483,E2 15423.483} C_VEL
LIN {X 0,Y 469.45,Z 1013.09,A -85,B 0,C 180,E1 15427.675,E2 15427.675} C_VEL
LIN {X 0,Y 478.933,Z 972.406,A -85,B 0,C 180,E1 15430.997,E2 15430.997} C_VEL
LIN {X 0,Y 487.449,Z 928.008,A -85,B 0,C 180,E1 15433.592,E2 15433.592} C_VEL
LIN {X 0,Y 492.768,Z 888.257,A -85,B 0,C 180,E1 15435.239,E2 15435.239} C_VEL
LIN {X 0,Y 478.201,Z 852.955,A -85,B 0,C 180,E1 15438.379,E2 15438.379} C_VEL
LIN {X 0,Y 458.603,Z 818.338,A -85,B 0,C 180,E1 15442.036,E2 15442.036} C_VEL
LIN {X 0,Y 439.302,Z 789.288,A -85,B 0,C 180,E1 15445.999,E2 15445.999} C_VEL
LIN {X 0,Y 436.627,Z 784.497,A -85,B 0,C 180,E1 15446.63,E2 15446.63} C_VEL
LIN {X 0,Y 436.55,Z 783.31,A -85,B 0,C 180,E1 15446.764,E2 15446.764} C_VEL
LIN {X 0,Y 436.823,Z 783.31,A -85,B 0,C 180,E1 15453.208,E2 15453.208} C_VEL
LIN {X 0,Y 437.052,Z 783.31,A -85,B 0,C 180,E1 15459.726,E2 15459.726} C_VEL
LIN {X 0,Y 437.295,Z 783.31,A -85,B 0,C 180,E1 15465.973,E2 15465.973} C_VEL
LIN {X 0,Y 437.649,Z 783.31,A -85,B 0,C 180,E1 15472.048,E2 15472.048} C_VEL
LIN {X 0,Y 438.01,Z 783.31,A -85,B 0,C 180,E1 15478.025,E2 15478.025} C_VEL
LIN {X 0,Y 437.926,Z 783.31,A -85,B 0,C 180,E1 15483.975,E2 15483.975} C_VEL
LIN {X 0,Y 437.551,Z 783.31,A -85,B 0,C 180,E1 15489.977,E2 15489.977} C_VEL
LIN {X 0,Y 437.221,Z 783.31,A -85,B 0,C 180,E1 15496.101,E2 15496.101} C_VEL
LIN {X 0,Y 436.92,Z 783.31,A -85,B 0,C 180,E1 15502.43,E2 15502.43} C_VEL
LIN {X 0,Y 436.612,Z 783.31,A -85,B 0,C 180,E1 15509.073,E2 15509.073} C_VEL
LIN {X 0,Y 436.431,Z 783.31,A -85,B 0,C 180,E1 15516.176,E2 15516.176} C_VEL
LIN {X 0,Y 436.447,Z 783.936,A -85,B 0,C 180,E1 15516.557,E2 15516.557} C_VEL
LIN {X 0,Y 439.007,Z 789.134,A -85,B 0,C 180,E1 15517.171,E2 15517.171} C_VEL
LIN {X 0,Y 453.053,Z 809.408,A -85,B 0,C 180,E1 15520.08,E2 15520.08} C_VEL
LIN {X 0,Y 474.631,Z 845.311,A -85,B 0,C 180,E1 15524.057,E2 15524.057} C_VEL
LIN {X 0,Y 491.025,Z 880.62,A -85,B 0,C 180,E1 15527.278,E2 15527.278} C_VEL
LIN {X 0,Y 493.339,Z 888.327,A -85,B 0,C 180,E1 15527.889,E2 15527.889} C_VEL
LIN {X 0,Y 487.079,Z 929.673,A -85,B 0,C 180,E1 15529.555,E2 15529.555} C_VEL
LIN {X 0,Y 479.189,Z 968.927,A -85,B 0,C 180,E1 15531.891,E2 15531.891} C_VEL
LIN {X 0,Y 470.443,Z 1004.972,A -85,B 0,C 180,E1 15534.873,E2 15534.873} C_VEL
LIN {X 0,Y 461.05,Z 1038.974,A -85,B 0,C 180,E1 15538.703,E2 15538.703} C_VEL
LIN {X 0,Y 452.689,Z 1067.972,A -85,B 0,C 180,E1 15543.14,E2 15543.14} C_VEL
LIN {X 0,Y 445.783,Z 1092.999,A -85,B 0,C 180,E1 15548.383,E2 15548.383} C_VEL
LIN {X 0,Y 441.335,Z 1112.078,A -85,B 0,C 180,E1 15554.061,E2 15554.061} C_VEL
LIN {X 0,Y 439.292,Z 1123.567,A -85,B 0,C 180,E1 15559.148,E2 15559.148} C_VEL
LIN {X 0,Y 438.527,Z 1130.405,A -85,B 0,C 180,E1 15564.052,E2 15564.052} C_VEL
LIN {X 0,Y 438.447,Z 1133.272,A -85,B 0,C 180,E1 15570.002,E2 15570.002} C_VEL
LIN {X 0,Y 438.54,Z 1130.32,A -85,B 0,C 180,E1 15575.951,E2 15575.951} C_VEL
LIN {X 0,Y 439.356,Z 1123.29,A -85,B 0,C 180,E1 15580.902,E2 15580.902} C_VEL
LIN {X 0,Y 441.667,Z 1110.484,A -85,B 0,C 180,E1 15586.391,E2 15586.391} C_VEL
LIN {X 0,Y 446.261,Z 1091.246,A -85,B 0,C 180,E1 15591.932,E2 15591.932} C_VEL
LIN {X 0,Y 452.838,Z 1067.415,A -85,B 0,C 180,E1 15596.855,E2 15596.855} C_VEL
LIN {X 0,Y 461.343,Z 1037.731,A -85,B 0,C 180,E1 15601.356,E2 15601.356} C_VEL
LIN {X 0,Y 470.637,Z 1003.795,A -85,B 0,C 180,E1 15605.144,E2 15605.144} C_VEL
LIN {X 0,Y 479.795,Z 965.894,A -85,B 0,C 180,E1 15608.228,E2 15608.228} C_VEL
LIN {X 0,Y 488.067,Z 924.16,A -85,B 0,C 180,E1 15610.611,E2 15610.611} C_VEL
LIN {X 0,Y 493.042,Z 885.936,A -85,B 0,C 180,E1 15612.147,E2 15612.147} C_VEL
LIN {X 0,Y 477.402,Z 850.443,A -85,B 0,C 180,E1 15615.34,E2 15615.34} C_VEL
LIN {X 0,Y 456.035,Z 814.067,A -85,B 0,C 180,E1 15619.221,E2 15619.221} C_VEL
LIN {X 0,Y 439.083,Z 789.246,A -85,B 0,C 180,E1 15622.685,E2 15622.685} C_VEL
LIN {X 0,Y 436.441,Z 784.22,A -85,B 0,C 180,E1 15623.309,E2 15623.309} C_VEL
LIN {X 0,Y 436.397,Z 783.31,A -85,B 0,C 180,E1 15623.446,E2 15623.446} C_VEL
LIN {X 0,Y 436.598,Z 783.31,A -85,B 0,C 180,E1 15630.184,E2 15630.184} C_VEL
LIN {X 0,Y 436.831,Z 783.31,A -85,B 0,C 180,E1 15635.398,E2 15635.398} C_VEL
LIN {X 0,Y 437.116,Z 783.31,A -85,B 0,C 180,E1 15641.816,E2 15641.816} C_VEL
LIN {X 0,Y 437.427,Z 783.31,A -85,B 0,C 180,E1 15647.998,E2 15647.998} C_VEL
LIN {X 0,Y 437.828,Z 783.31,A -85,B 0,C 180,E1 15654.034,E2 15654.034} C_VEL
LIN {X 0,Y 438.2,Z 783.31,A -85,B 0,C 180,E1 15659.993,E2 15659.993} C_VEL
LIN {X 0,Y 437.822,Z 783.31,A -85,B 0,C 180,E1 15665.951,E2 15665.951} C_VEL
LIN {X 0,Y 437.463,Z 783.31,A -85,B 0,C 180,E1 15671.985,E2 15671.985} C_VEL
LIN {X 0,Y 437.185,Z 783.31,A -85,B 0,C 180,E1 15678.165,E2 15678.165} C_VEL
LIN {X 0,Y 436.843,Z 783.31,A -85,B 0,C 180,E1 15684.585,E2 15684.585} C_VEL
LIN {X 0,Y 436.621,Z 783.31,A -85,B 0,C 180,E1 15691.356,E2 15691.356} C_VEL
LIN {X 0,Y 436.575,Z 783.62,A -85,B 0,C 180,E1 15693.372,E2 15693.372} C_VEL
LIN {X 0,Y 438.682,Z 788.695,A -85,B 0,C 180,E1 15693.907,E2 15693.907} C_VEL
LIN {X 0,Y 441.82,Z 793.174,A -85,B 0,C 180,E1 15694.597,E2 15694.597} C_VEL
LIN {X 0,Y 460.575,Z 821.772,A -85,B 0,C 180,E1 15698.371,E2 15698.371} C_VEL
LIN {X 0,Y 479.593,Z 856.192,A -85,B 0,C 180,E1 15701.928,E2 15701.928} C_VEL
LIN {X 0,Y 493.078,Z 889.247,A -85,B 0,C 180,E1 15704.857,E2 15704.857} C_VEL
LIN {X 0,Y 486.869,Z 930.94,A -85,B 0,C 180,E1 15706.567,E2 15706.567} C_VEL
LIN {X 0,Y 478.799,Z 972.669,A -85,B 0,C 180,E1 15709.028,E2 15709.028} C_VEL
LIN {X 0,Y 469.443,Z 1012.939,A -85,B 0,C 180,E1 15712.32,E2 15712.32} C_VEL
LIN {X 0,Y 459.821,Z 1050.635,A -85,B 0,C 180,E1 15716.512,E2 15716.512} C_VEL
LIN {X 0,Y 451.283,Z 1083.017,A -85,B 0,C 180,E1 15721.36,E2 15721.36} C_VEL
LIN {X 0,Y 444.9,Z 1109.999,A -85,B 0,C 180,E1 15726.825,E2 15726.825} C_VEL
LIN {X 0,Y 440.898,Z 1130.363,A -85,B 0,C 180,E1 15732.499,E2 15732.499} C_VEL
LIN {X 0,Y 439.035,Z 1144.225,A -85,B 0,C 180,E1 15738.048,E2 15738.048} C_VEL
LIN {X 0,Y 438.452,Z 1152.172,A -85,B 0,C 180,E1 15743.051,E2 15743.051} C_VEL
LIN {X 0,Y 438.291,Z 1155.915,A -85,B 0,C 180,E1 15748.017,E2 15748.017} C_VEL
LIN {X 0,Y 438.292,Z 1155.917,A -85,B 0,C 180,E1 15751.979,E2 15751.979} C_VEL
LIN {X 0,Y 438.427,Z 1152.183,A -85,B 0,C 180,E1 15756.946,E2 15756.946} C_VEL
LIN {X 0,Y 439.114,Z 1143.243,A -85,B 0,C 180,E1 15762.452,E2 15762.452} C_VEL
LIN {X 0,Y 440.96,Z 1130.356,A -85,B 0,C 180,E1 15767.509,E2 15767.509} C_VEL
LIN {X 0,Y 438.093,Z 1124.103,A -85,B 0,C 180,E1 15769.615,E2 15769.615} C_VEL
LIN {X 0,Y 435.771,Z 1117.19,A -85,B 0,C 180,E1 15771.707,E2 15771.707} C_VEL
LIN {X 0,Y 441.697,Z 1092.644,A -85,B 0,C 180,E1 15777.308,E2 15777.308} C_VEL
LIN {X 0,Y 449.493,Z 1062.823,A -85,B 0,C 180,E1 15782.35,E2 15782.35} C_VEL
LIN {X 0,Y 459.012,Z 1028.076,A -85,B 0,C 180,E1 15786.719,E2 15786.719} C_VEL
LIN {X 0,Y 468.248,Z 991.405,A -85,B 0,C 180,E1 15790.174,E2 15790.174} C_VEL
LIN {X 0,Y 476.948,Z 952.382,A -85,B 0,C 180,E1 15792.899,E2 15792.899} C_VEL
LIN {X 0,Y 484.59,Z 910.157,A -85,B 0,C 180,E1 15795.009,E2 15795.009} C_VEL
LIN {X 0,Y 486.783,Z 891.378,A -85,B 0,C 180,E1 15795.765,E2 15795.765} C_VEL
LIN {X 0,Y 472.784,Z 856.867,A -85,B 0,C 180,E1 15798.944,E2 15798.944} C_VEL
LIN {X 0,Y 454.703,Z 824.253,A -85,B 0,C 180,E1 15802.484,E2 15802.484} C_VEL
LIN {X 0,Y 435.81,Z 795.646,A -85,B 0,C 180,E1 15806.461,E2 15806.461} C_VEL
LIN {X 0,Y 431.25,Z 789.153,A -85,B 0,C 180,E1 15807.525,E2 15807.525} C_VEL
LIN {X 0,Y 428.736,Z 784.117,A -85,B 0,C 180,E1 15808.179,E2 15808.179} C_VEL
LIN {X 0,Y 428.828,Z 783.31,A -85,B 0,C 180,E1 15812.668,E2 15812.668} C_VEL
LIN {X 0,Y 429.13,Z 783.31,A -85,B 0,C 180,E1 15819.334,E2 15819.334} C_VEL
LIN {X 0,Y 429.38,Z 783.31,A -85,B 0,C 180,E1 15825.708,E2 15825.708} C_VEL
LIN {X 0,Y 429.723,Z 783.31,A -85,B 0,C 180,E1 15831.901,E2 15831.901} C_VEL
LIN {X 0,Y 430.103,Z 783.31,A -85,B 0,C 180,E1 15837.989,E2 15837.989} C_VEL
LIN {X 0,Y 430.011,Z 783.31,A -85,B 0,C 180,E1 15844.048,E2 15844.048} C_VEL
LIN {X 0,Y 429.628,Z 783.31,A -85,B 0,C 180,E1 15850.163,E2 15850.163} C_VEL
LIN {X 0,Y 429.265,Z 783.31,A -85,B 0,C 180,E1 15856.408,E2 15856.408} C_VEL
LIN {X 0,Y 428.899,Z 783.31,A -85,B 0,C 180,E1 15863.297,E2 15863.297} C_VEL
LIN {X 0,Y 428.699,Z 783.31,A -85,B 0,C 180,E1 15869.663,E2 15869.663} C_VEL
LIN {X 0,Y 428.482,Z 783.43,A -85,B 0,C 180,E1 15874.984,E2 15874.984} C_VEL
LIN {X 0,Y 430.645,Z 788.749,A -85,B 0,C 180,E1 15875.572,E2 15875.572} C_VEL
LIN {X 0,Y 433.389,Z 792.128,A -85,B 0,C 180,E1 15876.202,E2 15876.202} C_VEL
LIN {X 0,Y 452.375,Z 820.153,A -85,B 0,C 180,E1 15880.23,E2 15880.23} C_VEL
LIN {X 0,Y 472.779,Z 855.772,A -85,B 0,C 180,E1 15884.12,E2 15884.12} C_VEL
LIN {X 0,Y 487.409,Z 890.034,A -85,B 0,C 180,E1 15887.299,E2 15887.299} C_VEL
LIN {X 0,Y 480.943,Z 931.092,A -85,B 0,C 180,E1 15888.993,E2 15888.993} C_VEL
LIN {X 0,Y 472.857,Z 969.781,A -85,B 0,C 180,E1 15891.332,E2 15891.332} C_VEL
LIN {X 0,Y 463.711,Z 1006.094,A -85,B 0,C 180,E1 15894.387,E2 15894.387} C_VEL
LIN {X 0,Y 454.222,Z 1039.253,A -85,B 0,C 180,E1 15898.178,E2 15898.178} C_VEL
LIN {X 0,Y 445.38,Z 1068.679,A -85,B 0,C 180,E1 15902.751,E2 15902.751} C_VEL
LIN {X 0,Y 438.658,Z 1091.898,A -85,B 0,C 180,E1 15907.671,E2 15907.671} C_VEL
LIN {X 0,Y 433.94,Z 1110.857,A -85,B 0,C 180,E1 15913.26,E2 15913.26} C_VEL
LIN {X 0,Y 431.499,Z 1123.631,A -85,B 0,C 180,E1 15918.868,E2 15918.868} C_VEL
LIN {X 0,Y 430.638,Z 1130.614,A -85,B 0,C 180,E1 15923.943,E2 15923.943} C_VEL
LIN {X 0,Y 430.548,Z 1133.48,A -85,B 0,C 180,E1 15930.002,E2 15930.002} C_VEL
LIN {X 0,Y 430.652,Z 1130.529,A -85,B 0,C 180,E1 15936.061,E2 15936.061} C_VEL
LIN {X 0,Y 431.538,Z 1123.429,A -85,B 0,C 180,E1 15941.144,E2 15941.144} C_VEL
LIN {X 0,Y 433.999,Z 1110.561,A -85,B 0,C 180,E1 15946.741,E2 15946.741} C_VEL
LIN {X 0,Y 438.797,Z 1091.489,A -85,B 0,C 180,E1 15952.325,E2 15952.325} C_VEL
LIN {X 0,Y 445.621,Z 1067.818,A -85,B 0,C 180,E1 15957.299,E2 15957.299} C_VEL
LIN {X 0,Y 454.338,Z 1038.679,A -85,B 0,C 180,E1 15961.799,E2 15961.799} C_VEL
LIN {X 0,Y 463.924,Z 1005.002,A -85,B 0,C 180,E1 15965.627,E2 15965.627} C_VEL
LIN {X 0,Y 473.406,Z 967.126,A -85,B 0,C 180,E1 15968.766,E2 15968.766} C_VEL
LIN {X 0,Y 482.007,Z 925.36,A -85,B 0,C 180,E1 15971.192,E2 15971.192} C_VEL
LIN {X 0,Y 487.003,Z 888.795,A -85,B 0,C 180,E1 15972.699,E2 15972.699} C_VEL
LIN {X 0,Y 471.819,Z 853.881,A -85,B 0,C 180,E1 15975.959,E2 15975.959} C_VEL
LIN {X 0,Y 451.965,Z 819.683,A -85,B 0,C 180,E1 15979.726,E2 15979.726} C_VEL
LIN {X 0,Y 435.152,Z 795.002,A -85,B 0,C 180,E1 15983.257,E2 15983.257} C_VEL
LIN {X 0,Y 431.329,Z 789.395,A -85,B 0,C 180,E1 15984.144,E2 15984.144} C_VEL
LIN {X 0,Y 428.553,Z 784.472,A -85,B 0,C 180,E1 15984.836,E2 15984.836} C_VEL
LIN {X 0,Y 428.453,Z 783.31,A -85,B 0,C 180,E1 15985.02,E2 15985.02} C_VEL
LIN {X 0,Y 428.713,Z 783.31,A -85,B 0,C 180,E1 15990.338,E2 15990.338} C_VEL
LIN {X 0,Y 429.012,Z 783.31,A -85,B 0,C 180,E1 15997.133,E2 15997.133} C_VEL
LIN {X 0,Y 429.255,Z 783.31,A -85,B 0,C 180,E1 16003.591,E2 16003.591} C_VEL
LIN {X 0,Y 429.665,Z 783.31,A -85,B 0,C 180,E1 16009.838,E2 16009.838} C_VEL
LIN {X 0,Y 430.03,Z 783.31,A -85,B 0,C 180,E1 16015.952,E2 16015.952} C_VEL
LIN {X 0,Y 430.197,Z 783.31,A -85,B 0,C 180,E1 16022.011,E2 16022.011} C_VEL
LIN {X 0,Y 429.737,Z 783.31,A -85,B 0,C 180,E1 16028.099,E2 16028.099} C_VEL
LIN {X 0,Y 429.454,Z 783.31,A -85,B 0,C 180,E1 16034.289,E2 16034.289} C_VEL
LIN {X 0,Y 429.136,Z 783.31,A -85,B 0,C 180,E1 16040.665,E2 16040.665} C_VEL
LIN {X 0,Y 428.797,Z 783.31,A -85,B 0,C 180,E1 16047.334,E2 16047.334} C_VEL
LIN {X 0,Y 428.691,Z 783.31,A -85,B 0,C 180,E1 16051.822,E2 16051.822} C_VEL
LIN {X 0,Y 430.827,Z 788.743,A -85,B 0,C 180,E1 16052.421,E2 16052.421} C_VEL
LIN {X 0,Y 433.489,Z 792.175,A -85,B 0,C 180,E1 16053.038,E2 16053.038} C_VEL
LIN {X 0,Y 452.553,Z 820.778,A -85,B 0,C 180,E1 16057.122,E2 16057.122} C_VEL
LIN {X 0,Y 471.694,Z 854.93,A -85,B 0,C 180,E1 16060.866,E2 16060.866} C_VEL
LIN {X 0,Y 486.196,Z 889.746,A -85,B 0,C 180,E1 16064.107,E2 16064.107} C_VEL
LIN {X 0,Y 486.692,Z 894.783,A -85,B 0,C 180,E1 16064.404,E2 16064.404} C_VEL
LIN {X 0,Y 479.343,Z 939.479,A -85,B 0,C 180,E1 16066.37,E2 16066.37} C_VEL
LIN {X 0,Y 471.084,Z 979.307,A -85,B 0,C 180,E1 16068.904,E2 16068.904} C_VEL
LIN {X 0,Y 462.049,Z 1016.386,A -85,B 0,C 180,E1 16072.084,E2 16072.084} C_VEL
LIN {X 0,Y 452.536,Z 1052.068,A -85,B 0,C 180,E1 16076.176,E2 16076.176} C_VEL
LIN {X 0,Y 443.772,Z 1084.004,A -85,B 0,C 180,E1 16081.08,E2 16081.08} C_VEL
LIN {X 0,Y 437.423,Z 1109.75,A -85,B 0,C 180,E1 16086.405,E2 16086.405} C_VEL
LIN {X 0,Y 433.156,Z 1130.131,A -85,B 0,C 180,E1 16092.176,E2 16092.176} C_VEL
LIN {X 0,Y 431.197,Z 1144.006,A -85,B 0,C 180,E1 16097.827,E2 16097.827} C_VEL
LIN {X 0,Y 430.546,Z 1151.96,A -85,B 0,C 180,E1 16102.923,E2 16102.923} C_VEL
LIN {X 0,Y 430.387,Z 1155.708,A -85,B 0,C 180,E1 16107.981,E2 16107.981} C_VEL
LIN {X 0,Y 430.39,Z 1155.71,A -85,B 0,C 180,E1 16112.016,E2 16112.016} C_VEL
LIN {X 0,Y 430.52,Z 1151.972,A -85,B 0,C 180,E1 16117.074,E2 16117.074} C_VEL
LIN {X 0,Y 431.29,Z 1143.026,A -85,B 0,C 180,E1 16122.682,E2 16122.682} C_VEL
LIN {X 0,Y 433.448,Z 1128.582,A -85,B 0,C 180,E1 16128.335,E2 16128.335} C_VEL
LIN {X 0,Y 435.771,Z 1117.19,A -85,B 0,C 180,E1 16131.707,E2 16131.707} C_VEL
LIN {X 0,Y 435.471,Z 1113.393,A -85,B 0,C 180,E1 16132.742,E2 16132.742} C_VEL
LIN {X 0,Y 431.706,Z 1102.865,A -85,B 0,C 180,E1 16135.589,E2 16135.589} C_VEL
LIN {X 0,Y 431.893,Z 1101.756,A -85,B 0,C 180,E1 16135.84,E2 16135.84} C_VEL
LIN {X 0,Y 439.933,Z 1072.373,A -85,B 0,C 180,E1 16141.391,E2 16141.391} C_VEL
LIN {X 0,Y 449.536,Z 1038.46,A -85,B 0,C 180,E1 16146.117,E2 16146.117} C_VEL
LIN {X 0,Y 460.058,Z 999.509,A -85,B 0,C 180,E1 16150.109,E2 16150.109} C_VEL
LIN {X 0,Y 469.898,Z 957.78,A -85,B 0,C 180,E1 16153.215,E2 16153.215} C_VEL
LIN {X 0,Y 478.027,Z 915.091,A -85,B 0,C 180,E1 16155.452,E2 16155.452} C_VEL
LIN {X 0,Y 480.873,Z 894.438,A -85,B 0,C 180,E1 16156.303,E2 16156.303} C_VEL
LIN {X 0,Y 467.184,Z 860.195,A -85,B 0,C 180,E1 16159.575,E2 16159.575} C_VEL
LIN {X 0,Y 448.577,Z 826.298,A -85,B 0,C 180,E1 16163.402,E2 16163.402} C_VEL
LIN {X 0,Y 428.556,Z 796.163,A -85,B 0,C 180,E1 16167.848,E2 16167.848} C_VEL
LIN {X 0,Y 423.619,Z 789.343,A -85,B 0,C 180,E1 16169.072,E2 16169.072} C_VEL
LIN {X 0,Y 420.912,Z 784.572,A -85,B 0,C 180,E1 16169.81,E2 16169.81} C_VEL
LIN {X 0,Y 420.823,Z 783.31,A -85,B 0,C 180,E1 16170.02,E2 16170.02} C_VEL
LIN {X 0,Y 421.107,Z 783.31,A -85,B 0,C 180,E1 16176.696,E2 16176.696} C_VEL
LIN {X 0,Y 421.35,Z 783.31,A -85,B 0,C 180,E1 16183.291,E2 16183.291} C_VEL
LIN {X 0,Y 421.708,Z 783.31,A -85,B 0,C 180,E1 16189.66,E2 16189.66} C_VEL
LIN {X 0,Y 422.127,Z 783.31,A -85,B 0,C 180,E1 16195.891,E2 16195.891} C_VEL
LIN {X 0,Y 422.286,Z 783.31,A -85,B 0,C 180,E1 16202.064,E2 16202.064} C_VEL
LIN {X 0,Y 421.812,Z 783.31,A -85,B 0,C 180,E1 16208.268,E2 16208.268} C_VEL
LIN {X 0,Y 421.471,Z 783.31,A -85,B 0,C 180,E1 16214.582,E2 16214.582} C_VEL
LIN {X 0,Y 421.129,Z 783.31,A -85,B 0,C 180,E1 16221.093,E2 16221.093} C_VEL
LIN {X 0,Y 420.807,Z 783.31,A -85,B 0,C 180,E1 16227.916,E2 16227.916} C_VEL
LIN {X 0,Y 420.603,Z 784.075,A -85,B 0,C 180,E1 16233.338,E2 16233.338} C_VEL
LIN {X 0,Y 423.135,Z 789.144,A -85,B 0,C 180,E1 16234.041,E2 16234.041} C_VEL
LIN {X 0,Y 426.01,Z 792.959,A -85,B 0,C 180,E1 16234.756,E2 16234.756} C_VEL
LIN {X 0,Y 442.291,Z 816.339,A -85,B 0,C 180,E1 16238.466,E2 16238.466} C_VEL
LIN {X 0,Y 463.027,Z 850.799,A -85,B 0,C 180,E1 16242.611,E2 16242.611} C_VEL
LIN {X 0,Y 478.796,Z 885.807,A -85,B 0,C 180,E1 16246.078,E2 16246.078} C_VEL
LIN {X 0,Y 481.305,Z 893.863,A -85,B 0,C 180,E1 16246.768,E2 16246.768} C_VEL
LIN {X 0,Y 474.076,Z 936.558,A -85,B 0,C 180,E1 16248.624,E2 16248.624} C_VEL
LIN {X 0,Y 465.156,Z 976.248,A -85,B 0,C 180,E1 16251.17,E2 16251.17} C_VEL
LIN {X 0,Y 455.819,Z 1011.285,A -85,B 0,C 180,E1 16254.306,E2 16254.306} C_VEL
LIN {X 0,Y 446.545,Z 1042.309,A -85,B 0,C 180,E1 16258.029,E2 16258.029} C_VEL
LIN {X 0,Y 437.732,Z 1070.511,A -85,B 0,C 180,E1 16262.575,E2 16262.575} C_VEL
LIN {X 0,Y 430.636,Z 1094.147,A -85,B 0,C 180,E1 16267.778,E2 16267.778} C_VEL
LIN {X 0,Y 425.937,Z 1112.518,A -85,B 0,C 180,E1 16273.468,E2 16273.468} C_VEL
LIN {X 0,Y 423.663,Z 1123.844,A -85,B 0,C 180,E1 16278.658,E2 16278.658} C_VEL
LIN {X 0,Y 422.749,Z 1130.822,A -85,B 0,C 180,E1 16283.829,E2 16283.829} C_VEL
LIN {X 0,Y 422.652,Z 1133.687,A -85,B 0,C 180,E1 16290.002,E2 16290.002} C_VEL
LIN {X 0,Y 422.608,Z 1132.374,A -85,B 0,C 180,E1 16294.114,E2 16294.114} C_VEL
LIN {X 0,Y 423.238,Z 1126.977,A -85,B 0,C 180,E1 16299.272,E2 16299.272} C_VEL
LIN {X 0,Y 424.878,Z 1117.407,A -85,B 0,C 180,E1 16304.457,E2 16304.457} C_VEL
LIN {X 0,Y 428.705,Z 1101.24,A -85,B 0,C 180,E1 16310.159,E2 16310.159} C_VEL
LIN {X 0,Y 434.939,Z 1079.481,A -85,B 0,C 180,E1 16315.539,E2 16315.539} C_VEL
LIN {X 0,Y 443.144,Z 1053.094,A -85,B 0,C 180,E1 16320.288,E2 16320.288} C_VEL
LIN {X 0,Y 452.235,Z 1023.262,A -85,B 0,C 180,E1 16324.285,E2 16324.285} C_VEL
LIN {X 0,Y 461.827,Z 989.3,A -85,B 0,C 180,E1 16327.667,E2 16327.667} C_VEL
LIN {X 0,Y 470.899,Z 951.564,A -85,B 0,C 180,E1 16330.42,E2 16330.42} C_VEL
LIN {X 0,Y 478.855,Z 909.588,A -85,B 0,C 180,E1 16332.547,E2 16332.547} C_VEL
LIN {X 0,Y 481.055,Z 891.891,A -85,B 0,C 180,E1 16333.247,E2 16333.247} C_VEL
LIN {X 0,Y 466.347,Z 857.428,A -85,B 0,C 180,E1 16336.577,E2 16336.577} C_VEL
LIN {X 0,Y 447.419,Z 824.466,A -85,B 0,C 180,E1 16340.342,E2 16340.342} C_VEL
LIN {X 0,Y 428.503,Z 796.278,A -85,B 0,C 180,E1 16344.507,E2 16344.507} C_VEL
LIN {X 0,Y 423.397,Z 789.351,A -85,B 0,C 180,E1 16345.76,E2 16345.76} C_VEL
LIN {X 0,Y 420.628,Z 784.242,A -85,B 0,C 180,E1 16346.514,E2 16346.514} C_VEL
LIN {X 0,Y 420.56,Z 783.31,A -85,B 0,C 180,E1 16346.663,E2 16346.663} C_VEL
LIN {X 0,Y 420.831,Z 783.31,A -85,B 0,C 180,E1 16352.086,E2 16352.086} C_VEL
LIN {X 0,Y 421.229,Z 783.31,A -85,B 0,C 180,E1 16359.269,E2 16359.269} C_VEL
LIN {X 0,Y 421.485,Z 783.31,A -85,B 0,C 180,E1 16366.08,E2 16366.08} C_VEL
LIN {X 0,Y 421.841,Z 783.31,A -85,B 0,C 180,E1 16372.249,E2 16372.249} C_VEL
LIN {X 0,Y 422.248,Z 783.31,A -85,B 0,C 180,E1 16377.936,E2 16377.936} C_VEL
LIN {X 0,Y 422.14,Z 783.31,A -85,B 0,C 180,E1 16384.108,E2 16384.108} C_VEL
LIN {X 0,Y 421.737,Z 783.31,A -85,B 0,C 180,E1 16390.34,E2 16390.34} C_VEL
LIN {X 0,Y 421.408,Z 783.31,A -85,B 0,C 180,E1 16396.707,E2 16396.707} C_VEL
LIN {X 0,Y 421.084,Z 783.31,A -85,B 0,C 180,E1 16403.306,E2 16403.306} C_VEL
LIN {X 0,Y 420.83,Z 783.812,A -85,B 0,C 180,E1 16410.194,E2 16410.194} C_VEL
LIN {X 0,Y 423.166,Z 788.911,A -85,B 0,C 180,E1 16410.862,E2 16410.862} C_VEL
LIN {X 0,Y 425.923,Z 792.567,A -85,B 0,C 180,E1 16411.554,E2 16411.554} C_VEL
LIN {X 0,Y 442.705,Z 817.429,A -85,B 0,C 180,E1 16415.416,E2 16415.416} C_VEL
LIN {X 0,Y 461.054,Z 848.155,A -85,B 0,C 180,E1 16419.154,E2 16419.154} C_VEL
LIN {X 0,Y 476.452,Z 882.205,A -85,B 0,C 180,E1 16422.578,E2 16422.578} C_VEL
LIN {X 0,Y 480.956,Z 895.311,A -85,B 0,C 180,E1 16423.767,E2 16423.767} C_VEL
LIN {X 0,Y 473.334,Z 940.125,A -85,B 0,C 180,E1 16425.76,E2 16425.76} C_VEL
LIN {X 0,Y 464.533,Z 980.918,A -85,B 0,C 180,E1 16428.398,E2 16428.398} C_VEL
LIN {X 0,Y 455.445,Z 1016.749,A -85,B 0,C 180,E1 16431.525,E2 16431.525} C_VEL
LIN {X 0,Y 445.776,Z 1051.774,A -85,B 0,C 180,E1 16435.591,E2 16435.591} C_VEL
LIN {X 0,Y 436.928,Z 1082.852,A -85,B 0,C 180,E1 16440.4,E2 16440.4} C_VEL
LIN {X 0,Y 430.055,Z 1109.037,A -85,B 0,C 180,E1 16445.861,E2 16445.861} C_VEL
LIN {X 0,Y 425.698,Z 1128.315,A -85,B 0,C 180,E1 16451.315,E2 16451.315} C_VEL
LIN {X 0,Y 423.458,Z 1142.788,A -85,B 0,C 180,E1 16457.076,E2 16457.076} C_VEL
LIN {X 0,Y 422.667,Z 1151.748,A -85,B 0,C 180,E1 16462.79,E2 16462.79} C_VEL
LIN {X 0,Y 422.503,Z 1155.501,A -85,B 0,C 180,E1 16467.943,E2 16467.943} C_VEL
LIN {X 0,Y 422.506,Z 1155.503,A -85,B 0,C 180,E1 16472.053,E2 16472.053} C_VEL
LIN {X 0,Y 422.641,Z 1151.761,A -85,B 0,C 180,E1 16477.206,E2 16477.206} C_VEL
LIN {X 0,Y 423.452,Z 1142.808,A -85,B 0,C 180,E1 16482.921,E2 16482.921} C_VEL
LIN {X 0,Y 425.75,Z 1128.353,A -85,B 0,C 180,E1 16488.679,E2 16488.679} C_VEL
LIN {X 0,Y 430.002,Z 1109.374,A -85,B 0,C 180,E1 16494.067,E2 16494.067} C_VEL
LIN {X 0,Y 431.893,Z 1101.756,A -85,B 0,C 180,E1 16495.84,E2 16495.84} C_VEL
LIN {X 0,Y 430.39,Z 1093.238,A -85,B 0,C 180,E1 16497.867,E2 16497.867} C_VEL
LIN {X 0,Y 429.348,Z 1084.106,A -85,B 0,C 180,E1 16499.868,E2 16499.868} C_VEL
LIN {X 0,Y 438.494,Z 1053.383,A -85,B 0,C 180,E1 16504.758,E2 16504.758} C_VEL
LIN {X 0,Y 448.251,Z 1019.516,A -85,B 0,C 180,E1 16508.814,E2 16508.814} C_VEL
LIN {X 0,Y 458.04,Z 982.52,A -85,B 0,C 180,E1 16512.139,E2 16512.139} C_VEL
LIN {X 0,Y 467.253,Z 941.755,A -85,B 0,C 180,E1 16514.825,E2 16514.825} C_VEL
LIN {X 0,Y 474.889,Z 897.259,A -85,B 0,C 180,E1 16516.873,E2 16516.873} C_VEL
LIN {X 0,Y 461.589,Z 863.493,A -85,B 0,C 180,E1 16520.23,E2 16520.23} C_VEL
LIN {X 0,Y 444.012,Z 831.113,A -85,B 0,C 180,E1 16524.028,E2 16524.028} C_VEL
LIN {X 0,Y 425.524,Z 802.856,A -85,B 0,C 180,E1 16528.255,E2 16528.255} C_VEL
LIN {X 0,Y 415.969,Z 789.486,A -85,B 0,C 180,E1 16530.76,E2 16530.76} C_VEL
LIN {X 0,Y 413.098,Z 784.664,A -85,B 0,C 180,E1 16531.601,E2 16531.601} C_VEL
LIN {X 0,Y 412.976,Z 783.31,A -85,B 0,C 180,E1 16531.703,E2 16531.703} C_VEL
LIN {X 0,Y 413.225,Z 783.31,A -85,B 0,C 180,E1 16538.5,E2 16538.5} C_VEL
LIN {X 0,Y 413.488,Z 783.31,A -85,B 0,C 180,E1 16545.147,E2 16545.147} C_VEL
LIN {X 0,Y 413.88,Z 783.31,A -85,B 0,C 180,E1 16551.588,E2 16551.588} C_VEL
LIN {X 0,Y 414.315,Z 783.31,A -85,B 0,C 180,E1 16557.912,E2 16557.912} C_VEL
LIN {X 0,Y 414.21,Z 783.31,A -85,B 0,C 180,E1 16564.203,E2 16564.203} C_VEL
LIN {X 0,Y 413.782,Z 783.31,A -85,B 0,C 180,E1 16570.557,E2 16570.557} C_VEL
LIN {X 0,Y 413.339,Z 783.31,A -85,B 0,C 180,E1 16577.629,E2 16577.629} C_VEL
LIN {X 0,Y 413.03,Z 783.31,A -85,B 0,C 180,E1 16583.805,E2 16583.805} C_VEL
LIN {X 0,Y 412.719,Z 783.31,A -85,B 0,C 180,E1 16590.934,E2 16590.934} C_VEL
LIN {X 0,Y 412.7,Z 783.453,A -85,B 0,C 180,E1 16591.492,E2 16591.492} C_VEL
LIN {X 0,Y 414.695,Z 788.595,A -85,B 0,C 180,E1 16592.136,E2 16592.136} C_VEL
LIN {X 0,Y 417.787,Z 792.118,A -85,B 0,C 180,E1 16592.962,E2 16592.962} C_VEL
LIN {X 0,Y 435.946,Z 818.219,A -85,B 0,C 180,E1 16597.388,E2 16597.388} C_VEL
LIN {X 0,Y 455.412,Z 850.245,A -85,B 0,C 180,E1 16601.479,E2 16601.479} C_VEL
LIN {X 0,Y 470.606,Z 882.866,A -85,B 0,C 180,E1 16604.905,E2 16604.905} C_VEL
LIN {X 0,Y 475.321,Z 896.651,A -85,B 0,C 180,E1 16606.188,E2 16606.188} C_VEL
LIN {X 0,Y 467.549,Z 940.276,A -85,B 0,C 180,E1 16608.16,E2 16608.16} C_VEL
LIN {X 0,Y 457.878,Z 981.066,A -85,B 0,C 180,E1 16610.893,E2 16610.893} C_VEL
LIN {X 0,Y 447.623,Z 1017.489,A -85,B 0,C 180,E1 16614.334,E2 16614.334} C_VEL
LIN {X 0,Y 437.711,Z 1049.197,A -85,B 0,C 180,E1 16618.43,E2 16618.43} C_VEL
LIN {X 0,Y 428.359,Z 1077.819,A -85,B 0,C 180,E1 16623.479,E2 16623.479} C_VEL
LIN {X 0,Y 421.289,Z 1101.102,A -85,B 0,C 180,E1 16629.25,E2 16629.25} C_VEL
LIN {X 0,Y 417.105,Z 1117.843,A -85,B 0,C 180,E1 16635.271,E2 16635.271} C_VEL
LIN {X 0,Y 415.152,Z 1128.769,A -85,B 0,C 180,E1 16641.607,E2 16641.607} C_VEL
LIN {X 0,Y 414.657,Z 1133.585,A -85,B 0,C 180,E1 16647.908,E2 16647.908} C_VEL
LIN {X 0,Y 414.718,Z 1133.561,A -85,B 0,C 180,E1 16652.096,E2 16652.096} C_VEL
LIN {X 0,Y 415.188,Z 1128.653,A -85,B 0,C 180,E1 16658.395,E2 16658.395} C_VEL
LIN {X 0,Y 417.134,Z 1117.625,A -85,B 0,C 180,E1 16664.732,E2 16664.732} C_VEL
LIN {X 0,Y 421.43,Z 1100.615,A -85,B 0,C 180,E1 16670.801,E2 16670.801} C_VEL
LIN {X 0,Y 428.537,Z 1077.344,A -85,B 0,C 180,E1 16676.513,E2 16676.513} C_VEL
LIN {X 0,Y 437.831,Z 1048.456,A -85,B 0,C 180,E1 16681.581,E2 16681.581} C_VEL
LIN {X 0,Y 448.122,Z 1015.707,A -85,B 0,C 180,E1 16685.755,E2 16685.755} C_VEL
LIN {X 0,Y 458.521,Z 978.543,A -85,B 0,C 180,E1 16689.198,E2 16689.198} C_VEL
LIN {X 0,Y 467.775,Z 939.019,A -85,B 0,C 180,E1 16691.807,E2 16691.807} C_VEL
LIN {X 0,Y 475.09,Z 894.75,A -85,B 0,C 180,E1 16693.828,E2 16693.828} C_VEL
LIN {X 0,Y 460.543,Z 860.164,A -85,B 0,C 180,E1 16697.294,E2 16697.294} C_VEL
LIN {X 0,Y 441.192,Z 826.343,A -85,B 0,C 180,E1 16701.342,E2 16701.342} C_VEL
LIN {X 0,Y 424.264,Z 801.516,A -85,B 0,C 180,E1 16705.217,E2 16705.217} C_VEL
LIN {X 0,Y 415.847,Z 789.623,A -85,B 0,C 180,E1 16707.419,E2 16707.419} C_VEL
LIN {X 0,Y 412.787,Z 784.509,A -85,B 0,C 180,E1 16708.304,E2 16708.304} C_VEL
LIN {X 0,Y 412.679,Z 783.31,A -85,B 0,C 180,E1 16708.38,E2 16708.38} C_VEL
LIN {X 0,Y 412.936,Z 783.31,A -85,B 0,C 180,E1 16713.87,E2 16713.87} C_VEL
LIN {X 0,Y 413.287,Z 783.31,A -85,B 0,C 180,E1 16720.728,E2 16720.728} C_VEL
LIN {X 0,Y 413.637,Z 783.31,A -85,B 0,C 180,E1 16727.297,E2 16727.297} C_VEL
LIN {X 0,Y 414.083,Z 783.31,A -85,B 0,C 180,E1 16733.69,E2 16733.69} C_VEL
LIN {X 0,Y 414.506,Z 783.31,A -85,B 0,C 180,E1 16739.992,E2 16739.992} C_VEL
LIN {X 0,Y 414.072,Z 783.31,A -85,B 0,C 180,E1 16746.294,E2 16746.294} C_VEL
LIN {X 0,Y 413.699,Z 783.31,A -85,B 0,C 180,E1 16752.685,E2 16752.685} C_VEL
LIN {X 0,Y 413.345,Z 783.31,A -85,B 0,C 180,E1 16759.253,E2 16759.253} C_VEL
LIN {X 0,Y 412.966,Z 783.31,A -85,B 0,C 180,E1 16766.11,E2 16766.11} C_VEL
LIN {X 0,Y 412.982,Z 783.973,A -85,B 0,C 180,E1 16768.405,E2 16768.405} C_VEL
LIN {X 0,Y 415.38,Z 789.016,A -85,B 0,C 180,E1 16769.142,E2 16769.142} C_VEL
LIN {X 0,Y 417.858,Z 791.844,A -85,B 0,C 180,E1 16769.799,E2 16769.799} C_VEL
LIN {X 0,Y 436.082,Z 818.765,A -85,B 0,C 180,E1 16774.287,E2 16774.287} C_VEL
LIN {X 0,Y 454.664,Z 849.875,A -85,B 0,C 180,E1 16778.276,E2 16778.276} C_VEL
LIN {X 0,Y 469.692,Z 882.935,A -85,B 0,C 180,E1 16781.762,E2 16781.762} C_VEL
LIN {X 0,Y 474.755,Z 899.154,A -85,B 0,C 180,E1 16783.24,E2 16783.24} C_VEL
LIN {X 0,Y 466.858,Z 943.267,A -85,B 0,C 180,E1 16785.266,E2 16785.266} C_VEL
LIN {X 0,Y 457.382,Z 985.202,A -85,B 0,C 180,E1 16788.08,E2 16788.08} C_VEL
LIN {X 0,Y 446.793,Z 1024.685,A -85,B 0,C 180,E1 16791.737,E2 16791.737} C_VEL
LIN {X 0,Y 436.92,Z 1058.646,A -85,B 0,C 180,E1 16795.998,E2 16795.998} C_VEL
LIN {X 0,Y 428.206,Z 1087.974,A -85,B 0,C 180,E1 16800.885,E2 16800.885} C_VEL
LIN {X 0,Y 421.901,Z 1111.508,A -85,B 0,C 180,E1 16806.095,E2 16806.095} C_VEL
LIN {X 0,Y 417.445,Z 1131.235,A -85,B 0,C 180,E1 16812.028,E2 16812.028} C_VEL
LIN {X 0,Y 415.286,Z 1145.566,A -85,B 0,C 180,E1 16818.422,E2 16818.422} C_VEL
LIN {X 0,Y 414.697,Z 1152.61,A -85,B 0,C 180,E1 16823.705,E2 16823.705} C_VEL
LIN {X 0,Y 414.706,Z 1155.648,A -85,B 0,C 180,E1 16829.998,E2 16829.998} C_VEL
LIN {X 0,Y 414.68,Z 1152.62,A -85,B 0,C 180,E1 16836.291,E2 16836.291} C_VEL
LIN {X 0,Y 415.252,Z 1145.587,A -85,B 0,C 180,E1 16841.575,E2 16841.575} C_VEL
LIN {X 0,Y 417.513,Z 1131.273,A -85,B 0,C 180,E1 16847.965,E2 16847.965} C_VEL
LIN {X 0,Y 422.341,Z 1110.031,A -85,B 0,C 180,E1 16854.301,E2 16854.301} C_VEL
LIN {X 0,Y 429.348,Z 1084.106,A -85,B 0,C 180,E1 16859.868,E2 16859.868} C_VEL
LIN {X 0,Y 428.652,Z 1074.517,A -85,B 0,C 180,E1 16861.828,E2 16861.828} C_VEL
LIN {X 0,Y 428.259,Z 1064.318,A -85,B 0,C 180,E1 16863.737,E2 16863.737} C_VEL
LIN {X 0,Y 437.862,Z 1032.989,A -85,B 0,C 180,E1 16867.95,E2 16867.95} C_VEL
LIN {X 0,Y 448.297,Z 996.548,A -85,B 0,C 180,E1 16871.642,E2 16871.642} C_VEL
LIN {X 0,Y 458.476,Z 955.863,A -85,B 0,C 180,E1 16874.659,E2 16874.659} C_VEL
LIN {X 0,Y 467.323,Z 911.618,A -85,B 0,C 180,E1 16876.959,E2 16876.959} C_VEL
LIN {X 0,Y 468.801,Z 899.831,A -85,B 0,C 180,E1 16877.475,E2 16877.475} C_VEL
LIN {X 0,Y 455.835,Z 866.422,A -85,B 0,C 180,E1 16880.929,E2 16880.929} C_VEL
LIN {X 0,Y 439.446,Z 835.848,A -85,B 0,C 180,E1 16884.661,E2 16884.661} C_VEL
LIN {X 0,Y 421.568,Z 808.387,A -85,B 0,C 180,E1 16888.904,E2 16888.904} C_VEL
LIN {X 0,Y 412.35,Z 795.493,A -85,B 0,C 180,E1 16891.403,E2 16891.403} C_VEL
LIN {X 0,Y 408.561,Z 789.902,A -85,B 0,C 180,E1 16892.527,E2 16892.527} C_VEL
LIN {X 0,Y 405.229,Z 784.878,A -85,B 0,C 180,E1 16893.576,E2 16893.576} C_VEL
LIN {X 0,Y 405.099,Z 783.31,A -85,B 0,C 180,E1 16893.847,E2 16893.847} C_VEL
LIN {X 0,Y 405.354,Z 783.31,A -85,B 0,C 180,E1 16900.352,E2 16900.352} C_VEL
LIN {X 0,Y 405.688,Z 783.31,A -85,B 0,C 180,E1 16907.06,E2 16907.06} C_VEL
LIN {X 0,Y 406.136,Z 783.31,A -85,B 0,C 180,E1 16913.583,E2 16913.583} C_VEL
LIN {X 0,Y 406.583,Z 783.31,A -85,B 0,C 180,E1 16920.008,E2 16920.008} C_VEL
LIN {X 0,Y 406.152,Z 783.31,A -85,B 0,C 180,E1 16926.433,E2 16926.433} C_VEL
LIN {X 0,Y 405.728,Z 783.31,A -85,B 0,C 180,E1 16932.955,E2 16932.955} C_VEL
LIN {X 0,Y 405.292,Z 783.31,A -85,B 0,C 180,E1 16939.668,E2 16939.668} C_VEL
LIN {X 0,Y 404.94,Z 783.31,A -85,B 0,C 180,E1 16946.686,E2 16946.686} C_VEL
LIN {X 0,Y 404.83,Z 783.803,A -85,B 0,C 180,E1 16949.507,E2 16949.507} C_VEL
LIN {X 0,Y 407.179,Z 788.978,A -85,B 0,C 180,E1 16950.306,E2 16950.306} C_VEL
LIN {X 0,Y 409.931,Z 791.906,A -85,B 0,C 180,E1 16951.1,E2 16951.1} C_VEL
LIN {X 0,Y 428.163,Z 817.742,A -85,B 0,C 180,E1 16955.904,E2 16955.904} C_VEL
LIN {X 0,Y 447.714,Z 849.35,A -85,B 0,C 180,E1 16960.259,E2 16960.259} C_VEL
LIN {X 0,Y 463.241,Z 881.892,A -85,B 0,C 180,E1 16963.879,E2 16963.879} C_VEL
LIN {X 0,Y 469.28,Z 900.021,A -85,B 0,C 180,E1 16965.634,E2 16965.634} C_VEL
LIN {X 0,Y 461.795,Z 940.356,A -85,B 0,C 180,E1 16967.486,E2 16967.486} C_VEL
LIN {X 0,Y 451.74,Z 981.418,A -85,B 0,C 180,E1 16970.258,E2 16970.258} C_VEL
LIN {X 0,Y 441.161,Z 1017.783,A -85,B 0,C 180,E1 16973.729,E2 16973.729} C_VEL
LIN {X 0,Y 430.968,Z 1049.167,A -85,B 0,C 180,E1 16977.826,E2 16977.826} C_VEL
LIN {X 0,Y 421.169,Z 1078.06,A -85,B 0,C 180,E1 16982.989,E2 16982.989} C_VEL
LIN {X 0,Y 414.068,Z 1100.299,A -85,B 0,C 180,E1 16988.538,E2 16988.538} C_VEL
LIN {X 0,Y 409.608,Z 1116.942,A -85,B 0,C 180,E1 16994.488,E2 16994.488} C_VEL
LIN {X 0,Y 407.544,Z 1127.095,A -85,B 0,C 180,E1 17000.044,E2 17000.044} C_VEL
LIN {X 0,Y 406.751,Z 1132.841,A -85,B 0,C 180,E1 17005.729,E2 17005.729} C_VEL
LIN {X 0,Y 406.876,Z 1134.1,A -85,B 0,C 180,E1 17010.002,E2 17010.002} C_VEL
LIN {X 0,Y 406.831,Z 1132.79,A -85,B 0,C 180,E1 17014.274,E2 17014.274} C_VEL
LIN {X 0,Y 407.593,Z 1126.922,A -85,B 0,C 180,E1 17019.976,E2 17019.976} C_VEL
LIN {X 0,Y 409.665,Z 1116.632,A -85,B 0,C 180,E1 17025.538,E2 17025.538} C_VEL
LIN {X 0,Y 414.21,Z 1099.941,A -85,B 0,C 180,E1 17031.458,E2 17031.458} C_VEL
LIN {X 0,Y 421.359,Z 1077.594,A -85,B 0,C 180,E1 17037.001,E2 17037.001} C_VEL
LIN {X 0,Y 430.891,Z 1049.087,A -85,B 0,C 180,E1 17042.089,E2 17042.089} C_VEL
LIN {X 0,Y 441.67,Z 1016.027,A -85,B 0,C 180,E1 17046.36,E2 17046.36} C_VEL
LIN {X 0,Y 452.384,Z 978.935,A -85,B 0,C 180,E1 17049.835,E2 17049.835} C_VEL
LIN {X 0,Y 462.154,Z 938.372,A -85,B 0,C 180,E1 17052.521,E2 17052.521} C_VEL
LIN {X 0,Y 469.173,Z 897.908,A -85,B 0,C 180,E1 17054.393,E2 17054.393} C_VEL
LIN {X 0,Y 455.251,Z 863.943,A -85,B 0,C 180,E1 17057.926,E2 17057.926} C_VEL
LIN {X 0,Y 437.275,Z 831.915,A -85,B 0,C 180,E1 17061.882,E2 17061.882} C_VEL
LIN {X 0,Y 420.132,Z 806.453,A -85,B 0,C 180,E1 17065.942,E2 17065.942} C_VEL
LIN {X 0,Y 412.187,Z 795.601,A -85,B 0,C 180,E1 17068.081,E2 17068.081} C_VEL
LIN {X 0,Y 408.263,Z 789.817,A -85,B 0,C 180,E1 17069.239,E2 17069.239} C_VEL
LIN {X 0,Y 405.093,Z 785.404,A -85,B 0,C 180,E1 17070.215,E2 17070.215} C_VEL
LIN {X 0,Y 404.828,Z 783.31,A -85,B 0,C 180,E1 17070.451,E2 17070.451} C_VEL
LIN {X 0,Y 405.102,Z 783.31,A -85,B 0,C 180,E1 17075.699,E2 17075.699} C_VEL
LIN {X 0,Y 405.469,Z 783.31,A -85,B 0,C 180,E1 17082.599,E2 17082.599} C_VEL
LIN {X 0,Y 405.863,Z 783.31,A -85,B 0,C 180,E1 17089.235,E2 17089.235} C_VEL
LIN {X 0,Y 406.31,Z 783.31,A -85,B 0,C 180,E1 17095.715,E2 17095.715} C_VEL
LIN {X 0,Y 406.49,Z 783.31,A -85,B 0,C 180,E1 17102.128,E2 17102.128} C_VEL
LIN {X 0,Y 406.005,Z 783.31,A -85,B 0,C 180,E1 17108.576,E2 17108.576} C_VEL
LIN {X 0,Y 405.605,Z 783.31,A -85,B 0,C 180,E1 17115.149,E2 17115.149} C_VEL
LIN {X 0,Y 405.261,Z 783.31,A -85,B 0,C 180,E1 17121.944,E2 17121.944} C_VEL
LIN {X 0,Y 405.054,Z 783.31,A -85,B 0,C 180,E1 17126.352,E2 17126.352} C_VEL
LIN {X 0,Y 407.147,Z 788.736,A -85,B 0,C 180,E1 17127.128,E2 17127.128} C_VEL
LIN {X 0,Y 410.331,Z 792.254,A -85,B 0,C 180,E1 17128.053,E2 17128.053} C_VEL
LIN {X 0,Y 427.549,Z 817.025,A -85,B 0,C 180,E1 17132.625,E2 17132.625} C_VEL
LIN {X 0,Y 446.999,Z 849.003,A -85,B 0,C 180,E1 17137.052,E2 17137.052} C_VEL
LIN {X 0,Y 462.27,Z 881.852,A -85,B 0,C 180,E1 17140.722,E2 17140.722} C_VEL
LIN {X 0,Y 468.819,Z 900.203,A -85,B 0,C 180,E1 17142.57,E2 17142.57} C_VEL
LIN {X 0,Y 460.731,Z 944.726,A -85,B 0,C 180,E1 17144.675,E2 17144.675} C_VEL
LIN {X 0,Y 450.745,Z 987.278,A -85,B 0,C 180,E1 17147.591,E2 17147.591} C_VEL
LIN {X 0,Y 439.859,Z 1026.387,A -85,B 0,C 180,E1 17151.301,E2 17151.301} C_VEL
LIN {X 0,Y 428.951,Z 1062.205,A -85,B 0,C 180,E1 17155.946,E2 17155.946} C_VEL
LIN {X 0,Y 419.957,Z 1091.796,A -85,B 0,C 180,E1 17161.145,E2 17161.145} C_VEL
LIN {X 0,Y 413.32,Z 1115.543,A -85,B 0,C 180,E1 17166.79,E2 17166.79} C_VEL
LIN {X 0,Y 409.172,Z 1133.779,A -85,B 0,C 180,E1 17172.766,E2 17172.766} C_VEL
LIN {X 0,Y 407.421,Z 1145.349,A -85,B 0,C 180,E1 17178.196,E2 17178.196} C_VEL
LIN {X 0,Y 406.827,Z 1152.401,A -85,B 0,C 180,E1 17183.583,E2 17183.583} C_VEL
LIN {X 0,Y 406.821,Z 1155.441,A -85,B 0,C 180,E1 17189.998,E2 17189.998} C_VEL
LIN {X 0,Y 406.674,Z 1154.077,A -85,B 0,C 180,E1 17194.271,E2 17194.271} C_VEL
LIN {X 0,Y 407.047,Z 1148.327,A -85,B 0,C 180,E1 17199.888,E2 17199.888} C_VEL
LIN {X 0,Y 408.745,Z 1136.429,A -85,B 0,C 180,E1 17206.2,E2 17206.2} C_VEL
LIN {X 0,Y 412.923,Z 1117.585,A -85,B 0,C 180,E1 17212.659,E2 17212.659} C_VEL
LIN {X 0,Y 420.004,Z 1091.875,A -85,B 0,C 180,E1 17218.847,E2 17218.847} C_VEL
LIN {X 0,Y 428.259,Z 1064.318,A -85,B 0,C 180,E1 17223.737,E2 17223.737} C_VEL
LIN {X 0,Y 428.192,Z 1053.685,A -85,B 0,C 180,E1 17225.606,E2 17225.606} C_VEL
LIN {X 0,Y 427.966,Z 1044.004,A -85,B 0,C 180,E1 17227.205,E2 17227.205} C_VEL
LIN {X 0,Y 428.395,Z 1042.477,A -85,B 0,C 180,E1 17227.409,E2 17227.409} C_VEL
LIN {X 0,Y 438.958,Z 1007.874,A -85,B 0,C 180,E1 17231.262,E2 17231.262} C_VEL
LIN {X 0,Y 449.298,Z 969.945,A -85,B 0,C 180,E1 17234.404,E2 17234.404} C_VEL
LIN {X 0,Y 458.699,Z 927.834,A -85,B 0,C 180,E1 17236.923,E2 17236.923} C_VEL
LIN {X 0,Y 462.738,Z 902.504,A -85,B 0,C 180,E1 17238.091,E2 17238.091} C_VEL
LIN {X 0,Y 450.425,Z 870.009,A -85,B 0,C 180,E1 17241.565,E2 17241.565} C_VEL
LIN {X 0,Y 434.009,Z 838.834,A -85,B 0,C 180,E1 17245.526,E2 17245.526} C_VEL
LIN {X 0,Y 415.144,Z 809.752,A -85,B 0,C 180,E1 17250.267,E2 17250.267} C_VEL
LIN {X 0,Y 405.289,Z 796.304,A -85,B 0,C 180,E1 17253.132,E2 17253.132} C_VEL
LIN {X 0,Y 400.929,Z 790.025,A -85,B 0,C 180,E1 17254.55,E2 17254.55} C_VEL
LIN {X 0,Y 397.509,Z 785.162,A -85,B 0,C 180,E1 17255.73,E2 17255.73} C_VEL
LIN {X 0,Y 397.262,Z 783.31,A -85,B 0,C 180,E1 17256.075,E2 17256.075} C_VEL
LIN {X 0,Y 397.533,Z 783.31,A -85,B 0,C 180,E1 17262.33,E2 17262.33} C_VEL
LIN {X 0,Y 397.932,Z 783.31,A -85,B 0,C 180,E1 17269.034,E2 17269.034} C_VEL
LIN {X 0,Y 398.371,Z 783.31,A -85,B 0,C 180,E1 17275.646,E2 17275.646} C_VEL
LIN {X 0,Y 398.558,Z 783.31,A -85,B 0,C 180,E1 17282.187,E2 17282.187} C_VEL
LIN {X 0,Y 398.06,Z 783.31,A -85,B 0,C 180,E1 17288.765,E2 17288.765} C_VEL
LIN {X 0,Y 397.62,Z 783.31,A -85,B 0,C 180,E1 17295.477,E2 17295.477} C_VEL
LIN {X 0,Y 397.207,Z 783.31,A -85,B 0,C 180,E1 17302.43,E2 17302.43} C_VEL
LIN {X 0,Y 396.979,Z 783.432,A -85,B 0,C 180,E1 17307.265,E2 17307.265} C_VEL
LIN {X 0,Y 398.752,Z 788.361,A -85,B 0,C 180,E1 17307.982,E2 17307.982} C_VEL
LIN {X 0,Y 402.221,Z 791.928,A -85,B 0,C 180,E1 17309.097,E2 17309.097} C_VEL
LIN {X 0,Y 418.131,Z 814.393,A -85,B 0,C 180,E1 17313.729,E2 17313.729} C_VEL
LIN {X 0,Y 435.407,Z 840.686,A -85,B 0,C 180,E1 17317.915,E2 17317.915} C_VEL
LIN {X 0,Y 451.867,Z 871.853,A -85,B 0,C 180,E1 17321.798,E2 17321.798} C_VEL
LIN {X 0,Y 463.288,Z 901.159,A -85,B 0,C 180,E1 17324.931,E2 17324.931} C_VEL
LIN {X 0,Y 455.685,Z 942.118,A -85,B 0,C 180,E1 17326.891,E2 17326.891} C_VEL
LIN {X 0,Y 445.654,Z 981.768,A -85,B 0,C 180,E1 17329.604,E2 17329.604} C_VEL
LIN {X 0,Y 434.602,Z 1018.468,A -85,B 0,C 180,E1 17333.151,E2 17333.151} C_VEL
LIN {X 0,Y 424.18,Z 1049.438,A -85,B 0,C 180,E1 17337.247,E2 17337.247} C_VEL
LIN {X 0,Y 414.022,Z 1078.298,A -85,B 0,C 180,E1 17342.484,E2 17342.484} C_VEL
LIN {X 0,Y 406.576,Z 1100.528,A -85,B 0,C 180,E1 17348.122,E2 17348.122} C_VEL
LIN {X 0,Y 401.89,Z 1117.161,A -85,B 0,C 180,E1 17354.183,E2 17354.183} C_VEL
LIN {X 0,Y 399.585,Z 1128.036,A -85,B 0,C 180,E1 17360.377,E2 17360.377} C_VEL
LIN {X 0,Y 398.855,Z 1133.049,A -85,B 0,C 180,E1 17365.645,E2 17365.645} C_VEL
LIN {X 0,Y 398.977,Z 1134.308,A -85,B 0,C 180,E1 17370.002,E2 17370.002} C_VEL
LIN {X 0,Y 398.933,Z 1132.998,A -85,B 0,C 180,E1 17374.358,E2 17374.358} C_VEL
LIN {X 0,Y 399.65,Z 1127.817,A -85,B 0,C 180,E1 17379.678,E2 17379.678} C_VEL
LIN {X 0,Y 401.96,Z 1116.853,A -85,B 0,C 180,E1 17385.843,E2 17385.843} C_VEL
LIN {X 0,Y 406.726,Z 1100.174,A -85,B 0,C 180,E1 17391.873,E2 17391.873} C_VEL
LIN {X 0,Y 414.173,Z 1077.843,A -85,B 0,C 180,E1 17397.509,E2 17397.509} C_VEL
LIN {X 0,Y 424.109,Z 1049.364,A -85,B 0,C 180,E1 17402.665,E2 17402.665} C_VEL
LIN {X 0,Y 435.093,Z 1016.912,A -85,B 0,C 180,E1 17406.922,E2 17406.922} C_VEL
LIN {X 0,Y 446.328,Z 979.323,A -85,B 0,C 180,E1 17410.487,E2 17410.487} C_VEL
LIN {X 0,Y 456.195,Z 939.684,A -85,B 0,C 180,E1 17413.147,E2 17413.147} C_VEL
LIN {X 0,Y 463.127,Z 900.561,A -85,B 0,C 180,E1 17415.013,E2 17415.013} C_VEL
LIN {X 0,Y 449.751,Z 867.173,A -85,B 0,C 180,E1 17418.623,E2 17418.623} C_VEL
LIN {X 0,Y 432.418,Z 835.981,A -85,B 0,C 180,E1 17422.649,E2 17422.649} C_VEL
LIN {X 0,Y 415.029,Z 809.801,A -85,B 0,C 180,E1 17426.962,E2 17426.962} C_VEL
LIN {X 0,Y 405.202,Z 796.423,A -85,B 0,C 180,E1 17429.793,E2 17429.793} C_VEL
LIN {X 0,Y 400.681,Z 790.029,A -85,B 0,C 180,E1 17431.243,E2 17431.243} C_VEL
LIN {X 0,Y 397.179,Z 785.167,A -85,B 0,C 180,E1 17432.441,E2 17432.441} C_VEL
LIN {X 0,Y 396.979,Z 783.31,A -85,B 0,C 180,E1 17432.735,E2 17432.735} C_VEL
LIN {X 0,Y 397.408,Z 783.31,A -85,B 0,C 180,E1 17439.925,E2 17439.925} C_VEL
LIN {X 0,Y 397.777,Z 783.31,A -85,B 0,C 180,E1 17446.781,E2 17446.781} C_VEL
LIN {X 0,Y 398.242,Z 783.31,A -85,B 0,C 180,E1 17453.438,E2 17453.438} C_VEL
LIN {X 0,Y 398.716,Z 783.31,A -85,B 0,C 180,E1 17459.992,E2 17459.992} C_VEL
LIN {X 0,Y 398.23,Z 783.31,A -85,B 0,C 180,E1 17466.545,E2 17466.545} C_VEL
LIN {X 0,Y 397.832,Z 783.31,A -85,B 0,C 180,E1 17473.2,E2 17473.2} C_VEL
LIN {X 0,Y 397.446,Z 783.31,A -85,B 0,C 180,E1 17480.055,E2 17480.055} C_VEL
LIN {X 0,Y 397.246,Z 783.658,A -85,B 0,C 180,E1 17484.203,E2 17484.203} C_VEL
LIN {X 0,Y 399.263,Z 788.638,A -85,B 0,C 180,E1 17484.995,E2 17484.995} C_VEL
LIN {X 0,Y 402.429,Z 791.925,A -85,B 0,C 180,E1 17486.004,E2 17486.004} C_VEL
LIN {X 0,Y 416.904,Z 812.565,A -85,B 0,C 180,E1 17490.27,E2 17490.27} C_VEL
LIN {X 0,Y 434.34,Z 839.535,A -85,B 0,C 180,E1 17494.595,E2 17494.595} C_VEL
LIN {X 0,Y 450.715,Z 871.009,A -85,B 0,C 180,E1 17498.556,E2 17498.556} C_VEL
LIN {X 0,Y 462.792,Z 902.916,A -85,B 0,C 180,E1 17501.963,E2 17501.963} C_VEL
LIN {X 0,Y 455.042,Z 944.573,A -85,B 0,C 180,E1 17503.974,E2 17503.974} C_VEL
LIN {X 0,Y 444.793,Z 986.909,A -85,B 0,C 180,E1 17506.886,E2 17506.886} C_VEL
LIN {X 0,Y 433.386,Z 1026.54,A -85,B 0,C 180,E1 17510.682,E2 17510.682} C_VEL
LIN {X 0,Y 422.378,Z 1061.521,A -85,B 0,C 180,E1 17515.264,E2 17515.264} C_VEL
LIN {X 0,Y 412.764,Z 1091.537,A -85,B 0,C 180,E1 17520.594,E2 17520.594} C_VEL
LIN {X 0,Y 405.533,Z 1116.484,A -85,B 0,C 180,E1 17526.66,E2 17526.66} C_VEL
LIN {X 0,Y 401.191,Z 1134.938,A -85,B 0,C 180,E1 17532.979,E2 17532.979} C_VEL
LIN {X 0,Y 399.359,Z 1146.84,A -85,B 0,C 180,E1 17539.063,E2 17539.063} C_VEL
LIN {X 0,Y 398.929,Z 1152.191,A -85,B 0,C 180,E1 17543.455,E2 17543.455} C_VEL
LIN {X 0,Y 398.809,Z 1154.879,A -85,B 0,C 180,E1 17547.821,E2 17547.821} C_VEL
LIN {X 0,Y 398.813,Z 1154.882,A -85,B 0,C 180,E1 17552.175,E2 17552.175} C_VEL
LIN {X 0,Y 398.993,Z 1151.129,A -85,B 0,C 180,E1 17557.636,E2 17557.636} C_VEL
LIN {X 0,Y 399.967,Z 1142.159,A -85,B 0,C 180,E1 17563.694,E2 17563.694} C_VEL
LIN {X 0,Y 402.741,Z 1127.671,A -85,B 0,C 180,E1 17569.789,E2 17569.789} C_VEL
LIN {X 0,Y 407.761,Z 1108.193,A -85,B 0,C 180,E1 17575.59,E2 17575.59} C_VEL
LIN {X 0,Y 415.849,Z 1082.063,A -85,B 0,C 180,E1 17581.278,E2 17581.278} C_VEL
LIN {X 0,Y 425.721,Z 1051.034,A -85,B 0,C 180,E1 17586.275,E2 17586.275} C_VEL
LIN {X 0,Y 428.395,Z 1042.477,A -85,B 0,C 180,E1 17587.409,E2 17587.409} C_VEL
LIN {X 0,Y 428.854,Z 1030.831,A -85,B 0,C 180,E1 17589.164,E2 17589.164} C_VEL
LIN {X 0,Y 429.019,Z 1020.319,A -85,B 0,C 180,E1 17590.662,E2 17590.662} C_VEL
LIN {X 0,Y 429.482,Z 1018.651,A -85,B 0,C 180,E1 17590.845,E2 17590.845} C_VEL
LIN {X 0,Y 440.138,Z 982.189,A -85,B 0,C 180,E1 17594.192,E2 17594.192} C_VEL
LIN {X 0,Y 450.326,Z 940.811,A -85,B 0,C 180,E1 17596.959,E2 17596.959} C_VEL
LIN {X 0,Y 457.063,Z 906.173,A -85,B 0,C 180,E1 17598.617,E2 17598.617} C_VEL
LIN {X 0,Y 445.263,Z 874.176,A -85,B 0,C 180,E1 17602.157,E2 17602.157} C_VEL
LIN {X 0,Y 429.542,Z 843.643,A -85,B 0,C 180,E1 17606.187,E2 17606.187} C_VEL
LIN {X 0,Y 412.002,Z 816.118,A -85,B 0,C 180,E1 17610.775,E2 17610.775} C_VEL
LIN {X 0,Y 398.415,Z 797.072,A -85,B 0,C 180,E1 17614.982,E2 17614.982} C_VEL
LIN {X 0,Y 394.624,Z 791.325,A -85,B 0,C 180,E1 17616.343,E2 17616.343} C_VEL
LIN {X 0,Y 389.784,Z 785.747,A -85,B 0,C 180,E1 17618.153,E2 17618.153} C_VEL
LIN {X 0,Y 389.41,Z 783.31,A -85,B 0,C 180,E1 17618.51,E2 17618.51} C_VEL
LIN {X 0,Y 389.651,Z 783.31,A -85,B 0,C 180,E1 17624.215,E2 17624.215} C_VEL
LIN {X 0,Y 390.147,Z 783.31,A -85,B 0,C 180,E1 17631.073,E2 17631.073} C_VEL
LIN {X 0,Y 390.595,Z 783.31,A -85,B 0,C 180,E1 17637.785,E2 17637.785} C_VEL
LIN {X 0,Y 390.646,Z 783.31,A -85,B 0,C 180,E1 17642.231,E2 17642.231} C_VEL
LIN {X 0,Y 390.125,Z 783.31,A -85,B 0,C 180,E1 17648.945,E2 17648.945} C_VEL
LIN {X 0,Y 389.673,Z 783.31,A -85,B 0,C 180,E1 17655.801,E2 17655.801} C_VEL
LIN {X 0,Y 389.283,Z 783.31,A -85,B 0,C 180,E1 17662.913,E2 17662.913} C_VEL
LIN {X 0,Y 389.223,Z 783.804,A -85,B 0,C 180,E1 17664.789,E2 17664.789} C_VEL
LIN {X 0,Y 391.425,Z 788.81,A -85,B 0,C 180,E1 17665.751,E2 17665.751} C_VEL
LIN {X 0,Y 394.577,Z 792.01,A -85,B 0,C 180,E1 17666.882,E2 17666.882} C_VEL
LIN {X 0,Y 409.475,Z 812.648,A -85,B 0,C 180,E1 17671.686,E2 17671.686} C_VEL
LIN {X 0,Y 427.546,Z 839.539,A -85,B 0,C 180,E1 17676.418,E2 17676.418} C_VEL
LIN {X 0,Y 444.415,Z 871.002,A -85,B 0,C 180,E1 17680.607,E2 17680.607} C_VEL
LIN {X 0,Y 456.838,Z 902.506,A -85,B 0,C 180,E1 17684.151,E2 17684.151} C_VEL
LIN {X 0,Y 457.002,Z 908.084,A -85,B 0,C 180,E1 17684.519,E2 17684.519} C_VEL
LIN {X 0,Y 448.856,Z 947.118,A -85,B 0,C 180,E1 17686.472,E2 17686.472} C_VEL
LIN {X 0,Y 438.838,Z 984.808,A -85,B 0,C 180,E1 17689.163,E2 17689.163} C_VEL
LIN {X 0,Y 428.161,Z 1019.007,A -85,B 0,C 180,E1 17692.541,E2 17692.541} C_VEL
LIN {X 0,Y 417.164,Z 1050.483,A -85,B 0,C 180,E1 17696.772,E2 17696.772} C_VEL
LIN {X 0,Y 406.894,Z 1078.535,A -85,B 0,C 180,E1 17701.96,E2 17701.96} C_VEL
LIN {X 0,Y 399.115,Z 1100.756,A -85,B 0,C 180,E1 17707.691,E2 17707.691} C_VEL
LIN {X 0,Y 394.14,Z 1117.616,A -85,B 0,C 180,E1 17713.969,E2 17713.969} C_VEL
LIN {X 0,Y 391.73,Z 1128.247,A -85,B 0,C 180,E1 17720.182,E2 17720.182} C_VEL
LIN {X 0,Y 390.96,Z 1133.256,A -85,B 0,C 180,E1 17725.556,E2 17725.556} C_VEL
LIN {X 0,Y 391.079,Z 1134.515,A -85,B 0,C 180,E1 17730.002,E2 17730.002} C_VEL
LIN {X 0,Y 391.035,Z 1133.206,A -85,B 0,C 180,E1 17734.447,E2 17734.447} C_VEL
LIN {X 0,Y 391.792,Z 1128.03,A -85,B 0,C 180,E1 17739.874,E2 17739.874} C_VEL
LIN {X 0,Y 394.207,Z 1117.295,A -85,B 0,C 180,E1 17746.065,E2 17746.065} C_VEL
LIN {X 0,Y 399.283,Z 1100.405,A -85,B 0,C 180,E1 17752.303,E2 17752.303} C_VEL
LIN {X 0,Y 407.054,Z 1078.089,A -85,B 0,C 180,E1 17758.032,E2 17758.032} C_VEL
LIN {X 0,Y 417.413,Z 1049.518,A -85,B 0,C 180,E1 17763.278,E2 17763.278} C_VEL
LIN {X 0,Y 429.086,Z 1016.089,A -85,B 0,C 180,E1 17767.688,E2 17767.688} C_VEL
LIN {X 0,Y 440.319,Z 979.709,A -85,B 0,C 180,E1 17771.158,E2 17771.158} C_VEL
LIN {X 0,Y 450.611,Z 939.543,A -85,B 0,C 180,E1 17773.869,E2 17773.869} C_VEL
LIN {X 0,Y 457.324,Z 903.969,A -85,B 0,C 180,E1 17775.577,E2 17775.577} C_VEL
LIN {X 0,Y 444.559,Z 871.292,A -85,B 0,C 180,E1 17779.235,E2 17779.235} C_VEL
LIN {X 0,Y 427.599,Z 839.836,A -85,B 0,C 180,E1 17783.429,E2 17783.429} C_VEL
LIN {X 0,Y 408.286,Z 810.733,A -85,B 0,C 180,E1 17788.52,E2 17788.52} C_VEL
LIN {X 0,Y 397.638,Z 796.639,A -85,B 0,C 180,E1 17791.856,E2 17791.856} C_VEL
LIN {X 0,Y 393.047,Z 790.149,A -85,B 0,C 180,E1 17793.504,E2 17793.504} C_VEL
LIN {X 0,Y 389.611,Z 785.831,A -85,B 0,C 180,E1 17794.808,E2 17794.808} C_VEL
LIN {X 0,Y 389.265,Z 783.31,A -85,B 0,C 180,E1 17795.208,E2 17795.208} C_VEL
LIN {X 0,Y 389.558,Z 783.31,A -85,B 0,C 180,E1 17801.864,E2 17801.864} C_VEL
LIN {X 0,Y 389.984,Z 783.31,A -85,B 0,C 180,E1 17808.791,E2 17808.791} C_VEL
LIN {X 0,Y 390.496,Z 783.31,A -85,B 0,C 180,E1 17815.541,E2 17815.541} C_VEL
LIN {X 0,Y 390.837,Z 783.31,A -85,B 0,C 180,E1 17819.992,E2 17819.992} C_VEL
LIN {X 0,Y 390.321,Z 783.31,A -85,B 0,C 180,E1 17826.679,E2 17826.679} C_VEL
LIN {X 0,Y 389.844,Z 783.31,A -85,B 0,C 180,E1 17833.669,E2 17833.669} C_VEL
LIN {X 0,Y 389.42,Z 783.31,A -85,B 0,C 180,E1 17840.96,E2 17840.96} C_VEL
LIN {X 0,Y 389.412,Z 784.12,A -85,B 0,C 180,E1 17841.735,E2 17841.735} C_VEL
LIN {X 0,Y 391.981,Z 789.18,A -85,B 0,C 180,E1 17842.81,E2 17842.81} C_VEL
LIN {X 0,Y 394.741,Z 791.84,A -85,B 0,C 180,E1 17843.79,E2 17843.79} C_VEL
LIN {X 0,Y 399.011,Z 797.524,A -85,B 0,C 180,E1 17845.278,E2 17845.278} C_VEL
LIN {X 0,Y 414.365,Z 819.839,A -85,B 0,C 180,E1 17849.945,E2 17849.945} C_VEL
LIN {X 0,Y 431.467,Z 847.011,A -85,B 0,C 180,E1 17854.324,E2 17854.324} C_VEL
LIN {X 0,Y 446.762,Z 877.9,A -85,B 0,C 180,E1 17858.287,E2 17858.287} C_VEL
LIN {X 0,Y 456.958,Z 906.128,A -85,B 0,C 180,E1 17861.39,E2 17861.39} C_VEL
LIN {X 0,Y 448.402,Z 948.585,A -85,B 0,C 180,E1 17863.5,E2 17863.5} C_VEL
LIN {X 0,Y 438.496,Z 987.951,A -85,B 0,C 180,E1 17866.283,E2 17866.283} C_VEL
LIN {X 0,Y 426.987,Z 1026.644,A -85,B 0,C 180,E1 17870.039,E2 17870.039} C_VEL
LIN {X 0,Y 415.69,Z 1061.242,A -85,B 0,C 180,E1 17874.622,E2 17874.622} C_VEL
LIN {X 0,Y 405.607,Z 1091.298,A -85,B 0,C 180,E1 17880.027,E2 17880.027} C_VEL
LIN {X 0,Y 398.329,Z 1115.123,A -85,B 0,C 180,E1 17885.879,E2 17885.879} C_VEL
LIN {X 0,Y 393.709,Z 1133.33,A -85,B 0,C 180,E1 17892.067,E2 17892.067} C_VEL
LIN {X 0,Y 391.742,Z 1144.915,A -85,B 0,C 180,E1 17897.716,E2 17897.716} C_VEL
LIN {X 0,Y 391.046,Z 1151.982,A -85,B 0,C 180,E1 17903.323,E2 17903.323} C_VEL
LIN {X 0,Y 390.933,Z 1154.672,A -85,B 0,C 180,E1 17907.777,E2 17907.777} C_VEL
LIN {X 0,Y 390.937,Z 1154.675,A -85,B 0,C 180,E1 17912.219,E2 17912.219} C_VEL
LIN {X 0,Y 391.102,Z 1150.918,A -85,B 0,C 180,E1 17917.791,E2 17917.791} C_VEL
LIN {X 0,Y 392.288,Z 1141.272,A -85,B 0,C 180,E1 17924.35,E2 17924.35} C_VEL
LIN {X 0,Y 395.46,Z 1125.861,A -85,B 0,C 180,E1 17930.755,E2 17930.755} C_VEL
LIN {X 0,Y 401.12,Z 1105.726,A -85,B 0,C 180,E1 17936.649,E2 17936.649} C_VEL
LIN {X 0,Y 409.323,Z 1080.315,A -85,B 0,C 180,E1 17942.146,E2 17942.146} C_VEL
LIN {X 0,Y 419.575,Z 1049.401,A -85,B 0,C 180,E1 17947.129,E2 17947.129} C_VEL
LIN {X 0,Y 429.482,Z 1018.651,A -85,B 0,C 180,E1 17950.845,E2 17950.845} C_VEL
LIN {X 0,Y 430.363,Z 1006.02,A -85,B 0,C 180,E1 17952.463,E2 17952.463} C_VEL
LIN {X 0,Y 431.086,Z 992.947,A -85,B 0,C 180,E1 17954.022,E2 17954.022} C_VEL
LIN {X 0,Y 441.527,Z 954.648,A -85,B 0,C 180,E1 17956.86,E2 17956.86} C_VEL
LIN {X 0,Y 450.844,Z 912.08,A -85,B 0,C 180,E1 17959.091,E2 17959.091} C_VEL
LIN {X 0,Y 450.364,Z 906.496,A -85,B 0,C 180,E1 17959.519,E2 17959.519} C_VEL
LIN {X 0,Y 439.085,Z 875.843,A -85,B 0,C 180,E1 17963.064,E2 17963.064} C_VEL
LIN {X 0,Y 423.17,Z 844.879,A -85,B 0,C 180,E1 17967.376,E2 17967.376} C_VEL
LIN {X 0,Y 405.26,Z 817.038,A -85,B 0,C 180,E1 17972.377,E2 17972.377} C_VEL
LIN {X 0,Y 394.811,Z 802.922,A -85,B 0,C 180,E1 17975.797,E2 17975.797} C_VEL
LIN {X 0,Y 390.675,Z 797.078,A -85,B 0,C 180,E1 17977.342,E2 17977.342} C_VEL
LIN {X 0,Y 386.935,Z 791.152,A -85,B 0,C 180,E1 17978.886,E2 17978.886} C_VEL
LIN {X 0,Y 382.019,Z 785.971,A -85,B 0,C 180,E1 17980.986,E2 17980.986} C_VEL
LIN {X 0,Y 381.615,Z 783.31,A -85,B 0,C 180,E1 17981.491,E2 17981.491} C_VEL
LIN {X 0,Y 382.039,Z 783.31,A -85,B 0,C 180,E1 17988.572,E2 17988.572} C_VEL
LIN {X 0,Y 382.553,Z 783.31,A -85,B 0,C 180,E1 17995.466,E2 17995.466} C_VEL
LIN {X 0,Y 382.899,Z 783.31,A -85,B 0,C 180,E1 18000.008,E2 18000.008} C_VEL
LIN {X 0,Y 382.379,Z 783.31,A -85,B 0,C 180,E1 18006.835,E2 18006.835} C_VEL
LIN {X 0,Y 381.926,Z 783.31,A -85,B 0,C 180,E1 18013.778,E2 18013.778} C_VEL
LIN {X 0,Y 381.466,Z 783.31,A -85,B 0,C 180,E1 18020.952,E2 18020.952} C_VEL
LIN {X 0,Y 381.411,Z 784.018,A -85,B 0,C 180,E1 18021.888,E2 18021.888} C_VEL
LIN {X 0,Y 383.702,Z 788.917,A -85,B 0,C 180,E1 18023.035,E2 18023.035} C_VEL
LIN {X 0,Y 386.974,Z 791.771,A -85,B 0,C 180,E1 18024.367,E2 18024.367} C_VEL
LIN {X 0,Y 390.957,Z 797.391,A -85,B 0,C 180,E1 18025.966,E2 18025.966} C_VEL
LIN {X 0,Y 406.36,Z 818.74,A -85,B 0,C 180,E1 18031.128,E2 18031.128} C_VEL
LIN {X 0,Y 424.35,Z 846.276,A -85,B 0,C 180,E1 18036.023,E2 18036.023} C_VEL
LIN {X 0,Y 440.229,Z 877.113,A -85,B 0,C 180,E1 18040.232,E2 18040.232} C_VEL
LIN {X 0,Y 451.435,Z 906.885,A -85,B 0,C 180,E1 18043.678,E2 18043.678} C_VEL
LIN {X 0,Y 443.241,Z 947.277,A -85,B 0,C 180,E1 18045.753,E2 18045.753} C_VEL
LIN {X 0,Y 433.237,Z 983.838,A -85,B 0,C 180,E1 18048.359,E2 18048.359} C_VEL
LIN {X 0,Y 421.861,Z 1019.296,A -85,B 0,C 180,E1 18051.882,E2 18051.882} C_VEL
LIN {X 0,Y 410.503,Z 1050.654,A -85,B 0,C 180,E1 18056.143,E2 18056.143} C_VEL
LIN {X 0,Y 399.816,Z 1078.77,A -85,B 0,C 180,E1 18061.418,E2 18061.418} C_VEL
LIN {X 0,Y 391.68,Z 1100.982,A -85,B 0,C 180,E1 18067.244,E2 18067.244} C_VEL
LIN {X 0,Y 386.443,Z 1117.834,A -85,B 0,C 180,E1 18073.64,E2 18073.64} C_VEL
LIN {X 0,Y 383.916,Z 1128.335,A -85,B 0,C 180,E1 18079.887,E2 18079.887} C_VEL
LIN {X 0,Y 383.066,Z 1133.464,A -85,B 0,C 180,E1 18085.465,E2 18085.465} C_VEL
LIN {X 0,Y 383.18,Z 1134.722,A -85,B 0,C 180,E1 18090.002,E2 18090.002} C_VEL
LIN {X 0,Y 383.139,Z 1133.414,A -85,B 0,C 180,E1 18094.538,E2 18094.538} C_VEL
LIN {X 0,Y 383.954,Z 1128.191,A -85,B 0,C 180,E1 18100.116,E2 18100.116} C_VEL
LIN {X 0,Y 386.515,Z 1117.515,A -85,B 0,C 180,E1 18106.394,E2 18106.394} C_VEL
LIN {X 0,Y 391.862,Z 1100.636,A -85,B 0,C 180,E1 18112.749,E2 18112.749} C_VEL
LIN {X 0,Y 399.961,Z 1078.334,A -85,B 0,C 180,E1 18118.575,E2 18118.575} C_VEL
LIN {X 0,Y 410.682,Z 1049.887,A -85,B 0,C 180,E1 18123.879,E2 18123.879} C_VEL
LIN {X 0,Y 422.819,Z 1016.403,A -85,B 0,C 180,E1 18128.347,E2 18128.347} C_VEL
LIN {X 0,Y 434.372,Z 980.085,A -85,B 0,C 180,E1 18131.847,E2 18131.847} C_VEL
LIN {X 0,Y 444.879,Z 940.274,A -85,B 0,C 180,E1 18134.56,E2 18134.56} C_VEL
LIN {X 0,Y 451.483,Z 906.981,A -85,B 0,C 180,E1 18136.192,E2 18136.192} C_VEL
LIN {X 0,Y 439.335,Z 875.281,A -85,B 0,C 180,E1 18139.881,E2 18139.881} C_VEL
LIN {X 0,Y 423.727,Z 845.408,A -85,B 0,C 180,E1 18143.995,E2 18143.995} C_VEL
LIN {X 0,Y 405.354,Z 817.298,A -85,B 0,C 180,E1 18149.023,E2 18149.023} C_VEL
LIN {X 0,Y 394.476,Z 802.784,A -85,B 0,C 180,E1 18152.547,E2 18152.547} C_VEL
LIN {X 0,Y 390.336,Z 797.008,A -85,B 0,C 180,E1 18154.081,E2 18154.081} C_VEL
LIN {X 0,Y 386.756,Z 791.221,A -85,B 0,C 180,E1 18155.549,E2 18155.549} C_VEL
LIN {X 0,Y 381.895,Z 786.021,A -85,B 0,C 180,E1 18157.62,E2 18157.62} C_VEL
LIN {X 0,Y 381.432,Z 783.31,A -85,B 0,C 180,E1 18158.014,E2 18158.014} C_VEL
LIN {X 0,Y 381.701,Z 783.31,A -85,B 0,C 180,E1 18163.86,E2 18163.86} C_VEL
LIN {X 0,Y 382.219,Z 783.31,A -85,B 0,C 180,E1 18170.869,E2 18170.869} C_VEL
LIN {X 0,Y 382.709,Z 783.31,A -85,B 0,C 180,E1 18177.723,E2 18177.723} C_VEL
LIN {X 0,Y 382.754,Z 783.31,A -85,B 0,C 180,E1 18182.26,E2 18182.26} C_VEL
LIN {X 0,Y 382.216,Z 783.31,A -85,B 0,C 180,E1 18189.114,E2 18189.114} C_VEL
LIN {X 0,Y 381.756,Z 783.31,A -85,B 0,C 180,E1 18196.12,E2 18196.12} C_VEL
LIN {X 0,Y 381.599,Z 783.323,A -85,B 0,C 180,E1 18198.81,E2 18198.81} C_VEL
LIN {X 0,Y 383.223,Z 788.183,A -85,B 0,C 180,E1 18199.702,E2 18199.702} C_VEL
LIN {X 0,Y 387.132,Z 791.944,A -85,B 0,C 180,E1 18201.317,E2 18201.317} C_VEL
LIN {X 0,Y 391.567,Z 797.722,A -85,B 0,C 180,E1 18203.054,E2 18203.054} C_VEL
LIN {X 0,Y 407.497,Z 820.523,A -85,B 0,C 180,E1 18208.363,E2 18208.363} C_VEL
LIN {X 0,Y 424.124,Z 846.697,A -85,B 0,C 180,E1 18212.922,E2 18212.922} C_VEL
LIN {X 0,Y 439.318,Z 876.685,A -85,B 0,C 180,E1 18217.05,E2 18217.05} C_VEL
LIN {X 0,Y 450.973,Z 908.718,A -85,B 0,C 180,E1 18220.735,E2 18220.735} C_VEL
LIN {X 0,Y 442.213,Z 950.938,A -85,B 0,C 180,E1 18222.913,E2 18222.913} C_VEL
LIN {X 0,Y 431.851,Z 990.336,A -85,B 0,C 180,E1 18225.776,E2 18225.776} C_VEL
LIN {X 0,Y 420.763,Z 1026.396,A -85,B 0,C 180,E1 18229.334,E2 18229.334} C_VEL
LIN {X 0,Y 408.779,Z 1061.76,A -85,B 0,C 180,E1 18234.086,E2 18234.086} C_VEL
LIN {X 0,Y 398.038,Z 1092.541,A -85,B 0,C 180,E1 18239.761,E2 18239.761} C_VEL
LIN {X 0,Y 390.339,Z 1116.806,A -85,B 0,C 180,E1 18245.938,E2 18245.938} C_VEL
LIN {X 0,Y 385.468,Z 1135.871,A -85,B 0,C 180,E1 18252.852,E2 18252.852} C_VEL
LIN {X 0,Y 383.651,Z 1146.412,A -85,B 0,C 180,E1 18258.609,E2 18258.609} C_VEL
LIN {X 0,Y 383.149,Z 1151.772,A -85,B 0,C 180,E1 18263.185,E2 18263.185} C_VEL
LIN {X 0,Y 383.026,Z 1154.465,A -85,B 0,C 180,E1 18267.731,E2 18267.731} C_VEL
LIN {X 0,Y 383.031,Z 1154.468,A -85,B 0,C 180,E1 18272.265,E2 18272.265} C_VEL
LIN {X 0,Y 383.231,Z 1149.752,A -85,B 0,C 180,E1 18278.82,E2 18278.82} C_VEL
LIN {X 0,Y 384.461,Z 1141.218,A -85,B 0,C 180,E1 18284.555,E2 18284.555} C_VEL
LIN {X 0,Y 387.865,Z 1125.636,A -85,B 0,C 180,E1 18291.181,E2 18291.181} C_VEL
LIN {X 0,Y 393.834,Z 1105.487,A -85,B 0,C 180,E1 18297.182,E2 18297.182} C_VEL
LIN {X 0,Y 402.382,Z 1080.055,A -85,B 0,C 180,E1 18302.769,E2 18302.769} C_VEL
LIN {X 0,Y 413.301,Z 1048.465,A -85,B 0,C 180,E1 18307.901,E2 18307.901} C_VEL
LIN {X 0,Y 425.277,Z 1012.512,A -85,B 0,C 180,E1 18312.183,E2 18312.183} C_VEL
LIN {X 0,Y 431.086,Z 992.947,A -85,B 0,C 180,E1 18314.022,E2 18314.022} C_VEL
LIN {X 0,Y 432.118,Z 979.383,A -85,B 0,C 180,E1 18315.499,E2 18315.499} C_VEL
LIN {X 0,Y 433.149,Z 965.378,A -85,B 0,C 180,E1 18316.887,E2 18316.887} C_VEL
LIN {X 0,Y 442.905,Z 924.817,A -85,B 0,C 180,E1 18319.26,E2 18319.26} C_VEL
LIN {X 0,Y 445.282,Z 911.853,A -85,B 0,C 180,E1 18319.894,E2 18319.894} C_VEL
LIN {X 0,Y 434.756,Z 881.674,A -85,B 0,C 180,E1 18323.471,E2 18323.471} C_VEL
LIN {X 0,Y 419.625,Z 851.064,A -85,B 0,C 180,E1 18327.838,E2 18327.838} C_VEL
LIN {X 0,Y 402.456,Z 823.674,A -85,B 0,C 180,E1 18332.852,E2 18332.852} C_VEL
LIN {X 0,Y 388.845,Z 804.548,A -85,B 0,C 180,E1 18337.607,E2 18337.607} C_VEL
LIN {X 0,Y 383.245,Z 797.328,A -85,B 0,C 180,E1 18339.923,E2 18339.923} C_VEL
LIN {X 0,Y 379.5,Z 791.766,A -85,B 0,C 180,E1 18341.7,E2 18341.7} C_VEL
LIN {X 0,Y 374.209,Z 785.802,A -85,B 0,C 180,E1 18344.451,E2 18344.451} C_VEL
LIN {X 0,Y 373.809,Z 783.31,A -85,B 0,C 180,E1 18345.035,E2 18345.035} C_VEL
LIN {X 0,Y 374.284,Z 783.31,A -85,B 0,C 180,E1 18350.691,E2 18350.691} C_VEL
LIN {X 0,Y 374.778,Z 783.31,A -85,B 0,C 180,E1 18357.692,E2 18357.692} C_VEL
LIN {X 0,Y 374.823,Z 783.31,A -85,B 0,C 180,E1 18362.325,E2 18362.325} C_VEL
LIN {X 0,Y 374.251,Z 783.31,A -85,B 0,C 180,E1 18369.327,E2 18369.327} C_VEL
LIN {X 0,Y 373.779,Z 783.31,A -85,B 0,C 180,E1 18376.492,E2 18376.492} C_VEL
LIN {X 0,Y 373.709,Z 783.789,A -85,B 0,C 180,E1 18378.384,E2 18378.384} C_VEL
LIN {X 0,Y 375.595,Z 788.585,A -85,B 0,C 180,E1 18379.6,E2 18379.6} C_VEL
LIN {X 0,Y 379.358,Z 791.888,A -85,B 0,C 180,E1 18381.458,E2 18381.458} C_VEL
LIN {X 0,Y 383.501,Z 797.64,A -85,B 0,C 180,E1 18383.385,E2 18383.385} C_VEL
LIN {X 0,Y 391.12,Z 808.327,A -85,B 0,C 180,E1 18386.479,E2 18386.479} C_VEL
LIN {X 0,Y 400.61,Z 821.351,A -85,B 0,C 180,E1 18389.738,E2 18389.738} C_VEL
LIN {X 0,Y 416.803,Z 845.704,A -85,B 0,C 180,E1 18394.459,E2 18394.459} C_VEL
LIN {X 0,Y 432.313,Z 874.93,A -85,B 0,C 180,E1 18398.789,E2 18398.789} C_VEL
LIN {X 0,Y 443.923,Z 904.499,A -85,B 0,C 180,E1 18402.436,E2 18402.436} C_VEL
LIN {X 0,Y 445.587,Z 912.152,A -85,B 0,C 180,E1 18403.196,E2 18403.196} C_VEL
LIN {X 0,Y 436.016,Z 954.168,A -85,B 0,C 180,E1 18405.428,E2 18405.428} C_VEL
LIN {X 0,Y 424.411,Z 993.752,A -85,B 0,C 180,E1 18408.499,E2 18408.499} C_VEL
LIN {X 0,Y 411.683,Z 1030.16,A -85,B 0,C 180,E1 18412.498,E2 18412.498} C_VEL
LIN {X 0,Y 399.739,Z 1061.48,A -85,B 0,C 180,E1 18417.324,E2 18417.324} C_VEL
LIN {X 0,Y 389.666,Z 1086.893,A -85,B 0,C 180,E1 18422.732,E2 18422.732} C_VEL
LIN {X 0,Y 381.963,Z 1107.938,A -85,B 0,C 180,E1 18429.085,E2 18429.085} C_VEL
LIN {X 0,Y 377.795,Z 1121.4,A -85,B 0,C 180,E1 18435.031,E2 18435.031} C_VEL
LIN {X 0,Y 375.884,Z 1129.816,A -85,B 0,C 180,E1 18440.723,E2 18440.723} C_VEL
LIN {X 0,Y 375.176,Z 1134.621,A -85,B 0,C 180,E1 18447.687,E2 18447.687} C_VEL
LIN {X 0,Y 375.251,Z 1134.598,A -85,B 0,C 180,E1 18452.316,E2 18452.316} C_VEL
LIN {X 0,Y 375.912,Z 1129.705,A -85,B 0,C 180,E1 18459.28,E2 18459.28} C_VEL
LIN {X 0,Y 378.543,Z 1118.71,A -85,B 0,C 180,E1 18466.273,E2 18466.273} C_VEL
LIN {X 0,Y 384.01,Z 1102.029,A -85,B 0,C 180,E1 18472.835,E2 18472.835} C_VEL
LIN {X 0,Y 392.416,Z 1079.757,A -85,B 0,C 180,E1 18478.86,E2 18478.86} C_VEL
LIN {X 0,Y 403.017,Z 1052.738,A -85,B 0,C 180,E1 18484.083,E2 18484.083} C_VEL
LIN {X 0,Y 414.69,Z 1021.957,A -85,B 0,C 180,E1 18488.401,E2 18488.401} C_VEL
LIN {X 0,Y 426.161,Z 987.978,A -85,B 0,C 180,E1 18491.901,E2 18491.901} C_VEL
LIN {X 0,Y 436.789,Z 950.773,A -85,B 0,C 180,E1 18494.678,E2 18494.678} C_VEL
LIN {X 0,Y 445.678,Z 910.028,A -85,B 0,C 180,E1 18496.824,E2 18496.824} C_VEL
LIN {X 0,Y 434.009,Z 878.713,A -85,B 0,C 180,E1 18500.598,E2 18500.598} C_VEL
LIN {X 0,Y 418.148,Z 848.005,A -85,B 0,C 180,E1 18505.037,E2 18505.037} C_VEL
LIN {X 0,Y 401.412,Z 822.553,A -85,B 0,C 180,E1 18509.851,E2 18509.851} C_VEL
LIN {X 0,Y 391.854,Z 809.402,A -85,B 0,C 180,E1 18513.078,E2 18513.078} C_VEL
LIN {X 0,Y 387.59,Z 803.642,A -85,B 0,C 180,E1 18514.7,E2 18514.7} C_VEL
LIN {X 0,Y 383.177,Z 797.37,A -85,B 0,C 180,E1 18516.56,E2 18516.56} C_VEL
LIN {X 0,Y 379.294,Z 791.577,A -85,B 0,C 180,E1 18518.384,E2 18518.384} C_VEL
LIN {X 0,Y 374.163,Z 786.084,A -85,B 0,C 180,E1 18521.014,E2 18521.014} C_VEL
LIN {X 0,Y 373.72,Z 783.31,A -85,B 0,C 180,E1 18521.511,E2 18521.511} C_VEL
LIN {X 0,Y 374.093,Z 783.31,A -85,B 0,C 180,E1 18528.308,E2 18528.308} C_VEL
LIN {X 0,Y 374.681,Z 783.31,A -85,B 0,C 180,E1 18535.353,E2 18535.353} C_VEL
LIN {X 0,Y 375.03,Z 783.31,A -85,B 0,C 180,E1 18539.991,E2 18539.991} C_VEL
LIN {X 0,Y 374.464,Z 783.31,A -85,B 0,C 180,E1 18546.963,E2 18546.963} C_VEL
LIN {X 0,Y 374.003,Z 783.31,A -85,B 0,C 180,E1 18554.058,E2 18554.058} C_VEL
LIN {X 0,Y 373.9,Z 783.959,A -85,B 0,C 180,E1 18555.412,E2 18555.412} C_VEL
LIN {X 0,Y 376.092,Z 788.847,A -85,B 0,C 180,E1 18556.767,E2 18556.767} C_VEL
LIN {X 0,Y 379.586,Z 791.953,A -85,B 0,C 180,E1 18558.458,E2 18558.458} C_VEL
LIN {X 0,Y 383.522,Z 797.514,A -85,B 0,C 180,E1 18560.288,E2 18560.288} C_VEL
LIN {X 0,Y 391.844,Z 809.196,A -85,B 0,C 180,E1 18563.64,E2 18563.64} C_VEL
LIN {X 0,Y 404.253,Z 826.494,A -85,B 0,C 180,E1 18567.774,E2 18567.774} C_VEL
LIN {X 0,Y 420.218,Z 852.3,A -85,B 0,C 180,E1 18572.388,E2 18572.388} C_VEL
LIN {X 0,Y 434.675,Z 881.902,A -85,B 0,C 180,E1 18576.563,E2 18576.563} C_VEL
LIN {X 0,Y 445.191,Z 911.79,A -85,B 0,C 180,E1 18580.116,E2 18580.116} C_VEL
LIN {X 0,Y 435.39,Z 956.226,A -85,B 0,C 180,E1 18582.493,E2 18582.493} C_VEL
LIN {X 0,Y 423.4,Z 998.972,A -85,B 0,C 180,E1 18585.804,E2 18585.804} C_VEL
LIN {X 0,Y 410.743,Z 1037.349,A -85,B 0,C 180,E1 18589.964,E2 18589.964} C_VEL
LIN {X 0,Y 398.636,Z 1071.019,A -85,B 0,C 180,E1 18594.986,E2 18594.986} C_VEL
LIN {X 0,Y 388.608,Z 1099.628,A -85,B 0,C 180,E1 18600.865,E2 18600.865} C_VEL
LIN {X 0,Y 381.317,Z 1121.987,A -85,B 0,C 180,E1 18607.204,E2 18607.204} C_VEL
LIN {X 0,Y 377.174,Z 1138.052,A -85,B 0,C 180,E1 18613.666,E2 18613.666} C_VEL
LIN {X 0,Y 375.574,Z 1147.823,A -85,B 0,C 180,E1 18619.538,E2 18619.538} C_VEL
LIN {X 0,Y 375.047,Z 1153.237,A -85,B 0,C 180,E1 18625.364,E2 18625.364} C_VEL
LIN {X 0,Y 375.224,Z 1154.612,A -85,B 0,C 180,E1 18629.998,E2 18629.998} C_VEL
LIN {X 0,Y 375.062,Z 1153.245,A -85,B 0,C 180,E1 18634.632,E2 18634.632} C_VEL
LIN {X 0,Y 375.539,Z 1147.846,A -85,B 0,C 180,E1 18640.459,E2 18640.459} C_VEL
LIN {X 0,Y 377.47,Z 1136.902,A -85,B 0,C 180,E1 18646.917,E2 18646.917} C_VEL
LIN {X 0,Y 381.856,Z 1120.252,A -85,B 0,C 180,E1 18653.375,E2 18653.375} C_VEL
LIN {X 0,Y 389.078,Z 1098.09,A -85,B 0,C 180,E1 18659.511,E2 18659.511} C_VEL
LIN {X 0,Y 398.576,Z 1071.176,A -85,B 0,C 180,E1 18665.008,E2 18665.008} C_VEL
LIN {X 0,Y 410.714,Z 1037.514,A -85,B 0,C 180,E1 18670.035,E2 18670.035} C_VEL
LIN {X 0,Y 423.432,Z 999.064,A -85,B 0,C 180,E1 18674.205,E2 18674.205} C_VEL
LIN {X 0,Y 433.149,Z 965.378,A -85,B 0,C 180,E1 18676.887,E2 18676.887} C_VEL
LIN {X 0,Y 434.095,Z 951.007,A -85,B 0,C 180,E1 18678.212,E2 18678.212} C_VEL
LIN {X 0,Y 434.92,Z 936.26,A -85,B 0,C 180,E1 18679.449,E2 18679.449} C_VEL
LIN {X 0,Y 439.3,Z 914.214,A -85,B 0,C 180,E1 18680.596,E2 18680.596} C_VEL
LIN {X 0,Y 428.949,Z 884.239,A -85,B 0,C 180,E1 18684.308,E2 18684.308} C_VEL
LIN {X 0,Y 415.089,Z 855.69,A -85,B 0,C 180,E1 18688.558,E2 18688.558} C_VEL
LIN {X 0,Y 399.486,Z 830.05,A -85,B 0,C 180,E1 18693.395,E2 18693.395} C_VEL
LIN {X 0,Y 386.337,Z 811.402,A -85,B 0,C 180,E1 18698.137,E2 18698.137} C_VEL
LIN {X 0,Y 381.028,Z 804.434,A -85,B 0,C 180,E1 18700.407,E2 18700.407} C_VEL
LIN {X 0,Y 376.301,Z 797.818,A -85,B 0,C 180,E1 18702.736,E2 18702.736} C_VEL
LIN {X 0,Y 372.286,Z 792.684,A -85,B 0,C 180,E1 18704.973,E2 18704.973} C_VEL
LIN {X 0,Y 370.951,Z 790.626,A -85,B 0,C 180,E1 18705.824,E2 18705.824} C_VEL
LIN {X 0,Y 366.695,Z 786.051,A -85,B 0,C 180,E1 18708.767,E2 18708.767} C_VEL
LIN {X 0,Y 366.241,Z 783.31,A -85,B 0,C 180,E1 18709.582,E2 18709.582} C_VEL
LIN {X 0,Y 366.732,Z 783.31,A -85,B 0,C 180,E1 18715.27,E2 18715.27} C_VEL
LIN {X 0,Y 367.092,Z 783.31,A -85,B 0,C 180,E1 18720.009,E2 18720.009} C_VEL
LIN {X 0,Y 366.506,Z 783.31,A -85,B 0,C 180,E1 18727.188,E2 18727.188} C_VEL
LIN {X 0,Y 366.141,Z 784.003,A -85,B 0,C 180,E1 18733.876,E2 18733.876} C_VEL
LIN {X 0,Y 368.026,Z 788.719,A -85,B 0,C 180,E1 18735.529,E2 18735.529} C_VEL
LIN {X 0,Y 371.919,Z 791.781,A -85,B 0,C 180,E1 18737.981,E2 18737.981} C_VEL
LIN {X 0,Y 375.11,Z 797.158,A -85,B 0,C 180,E1 18739.881,E2 18739.881} C_VEL
LIN {X 0,Y 377.587,Z 799.623,A -85,B 0,C 180,E1 18741.126,E2 18741.126} C_VEL
LIN {X 0,Y 383.795,Z 808.354,A -85,B 0,C 180,E1 18744.004,E2 18744.004} C_VEL
LIN {X 0,Y 393.711,Z 821.981,A -85,B 0,C 180,E1 18747.823,E2 18747.823} C_VEL
LIN {X 0,Y 408.508,Z 843.85,A -85,B 0,C 180,E1 18752.541,E2 18752.541} C_VEL
LIN {X 0,Y 423.602,Z 871.104,A -85,B 0,C 180,E1 18756.999,E2 18756.999} C_VEL
LIN {X 0,Y 436.365,Z 902.004,A -85,B 0,C 180,E1 18761.104,E2 18761.104} C_VEL
LIN {X 0,Y 439.907,Z 914.325,A -85,B 0,C 180,E1 18762.524,E2 18762.524} C_VEL
LIN {X 0,Y 430.106,Z 955.65,A -85,B 0,C 180,E1 18764.761,E2 18764.761} C_VEL
LIN {X 0,Y 418.36,Z 994.442,A -85,B 0,C 180,E1 18767.813,E2 18767.813} C_VEL
LIN {X 0,Y 405.994,Z 1028.909,A -85,B 0,C 180,E1 18771.608,E2 18771.608} C_VEL
LIN {X 0,Y 393.406,Z 1060.772,A -85,B 0,C 180,E1 18776.51,E2 18776.51} C_VEL
LIN {X 0,Y 382.408,Z 1087.408,A -85,B 0,C 180,E1 18782.256,E2 18782.256} C_VEL
LIN {X 0,Y 374.452,Z 1108.157,A -85,B 0,C 180,E1 18788.646,E2 18788.646} C_VEL
LIN {X 0,Y 369.996,Z 1121.828,A -85,B 0,C 180,E1 18794.825,E2 18794.825} C_VEL
LIN {X 0,Y 367.872,Z 1130.808,A -85,B 0,C 180,E1 18801.324,E2 18801.324} C_VEL
LIN {X 0,Y 367.273,Z 1134.828,A -85,B 0,C 180,E1 18807.638,E2 18807.638} C_VEL
LIN {X 0,Y 367.348,Z 1134.806,A -85,B 0,C 180,E1 18812.366,E2 18812.366} C_VEL
LIN {X 0,Y 368.061,Z 1129.916,A -85,B 0,C 180,E1 18819.48,E2 18819.48} C_VEL
LIN {X 0,Y 370.861,Z 1118.926,A -85,B 0,C 180,E1 18826.62,E2 18826.62} C_VEL
LIN {X 0,Y 376.379,Z 1102.828,A -85,B 0,C 180,E1 18833.112,E2 18833.112} C_VEL
LIN {X 0,Y 384.887,Z 1081.171,A -85,B 0,C 180,E1 18839.156,E2 18839.156} C_VEL
LIN {X 0,Y 395.254,Z 1055.84,A -85,B 0,C 180,E1 18844.244,E2 18844.244} C_VEL
LIN {X 0,Y 407.212,Z 1025.579,A -85,B 0,C 180,E1 18848.689,E2 18848.689} C_VEL
LIN {X 0,Y 419.419,Z 991.011,A -85,B 0,C 180,E1 18852.39,E2 18852.39} C_VEL
LIN {X 0,Y 430.863,Z 952.6,A -85,B 0,C 180,E1 18855.332,E2 18855.332} C_VEL
LIN {X 0,Y 439.719,Z 912.439,A -85,B 0,C 180,E1 18857.53,E2 18857.53} C_VEL
LIN {X 0,Y 428.231,Z 881.238,A -85,B 0,C 180,E1 18861.47,E2 18861.47} C_VEL
LIN {X 0,Y 413.479,Z 852.129,A -85,B 0,C 180,E1 18865.861,E2 18865.861} C_VEL
LIN {X 0,Y 396.051,Z 824.926,A -85,B 0,C 180,E1 18871.222,E2 18871.222} C_VEL
LIN {X 0,Y 385.251,Z 810.522,A -85,B 0,C 180,E1 18875.192,E2 18875.192} C_VEL
LIN {X 0,Y 380.904,Z 804.429,A -85,B 0,C 180,E1 18877.076,E2 18877.076} C_VEL
LIN {X 0,Y 376.126,Z 797.81,A -85,B 0,C 180,E1 18879.4,E2 18879.4} C_VEL
LIN {X 0,Y 372.169,Z 792.705,A -85,B 0,C 180,E1 18881.594,E2 18881.594} C_VEL
LIN {X 0,Y 371.136,Z 790.779,A -85,B 0,C 180,E1 18882.261,E2 18882.261} C_VEL
LIN {X 0,Y 366.562,Z 786.37,A -85,B 0,C 180,E1 18885.327,E2 18885.327} C_VEL
LIN {X 0,Y 366.051,Z 783.31,A -85,B 0,C 180,E1 18885.996,E2 18885.996} C_VEL
LIN {X 0,Y 366.561,Z 783.31,A -85,B 0,C 180,E1 18892.869,E2 18892.869} C_VEL
LIN {X 0,Y 367.126,Z 783.31,A -85,B 0,C 180,E1 18899.991,E2 18899.991} C_VEL
LIN {X 0,Y 366.521,Z 783.31,A -85,B 0,C 180,E1 18907.175,E2 18907.175} C_VEL
LIN {X 0,Y 366.256,Z 783.954,A -85,B 0,C 180,E1 18910.945,E2 18910.945} C_VEL
LIN {X 0,Y 368.642,Z 789.094,A -85,B 0,C 180,E1 18912.913,E2 18912.913} C_VEL
LIN {X 0,Y 372.107,Z 792.021,A -85,B 0,C 180,E1 18915.035,E2 18915.035} C_VEL
LIN {X 0,Y 375.776,Z 797.477,A -85,B 0,C 180,E1 18917.138,E2 18917.138} C_VEL
LIN {X 0,Y 377.839,Z 799.922,A -85,B 0,C 180,E1 18918.171,E2 18918.171} C_VEL
LIN {X 0,Y 383.717,Z 808.077,A -85,B 0,C 180,E1 18920.881,E2 18920.881} C_VEL
LIN {X 0,Y 392.975,Z 820.827,A -85,B 0,C 180,E1 18924.475,E2 18924.475} C_VEL
LIN {X 0,Y 407.541,Z 842.636,A -85,B 0,C 180,E1 18929.208,E2 18929.208} C_VEL
LIN {X 0,Y 423.442,Z 872.183,A -85,B 0,C 180,E1 18934.026,E2 18934.026} C_VEL
LIN {X 0,Y 435.591,Z 902.604,A -85,B 0,C 180,E1 18938.039,E2 18938.039} C_VEL
LIN {X 0,Y 439.205,Z 916.156,A -85,B 0,C 180,E1 18939.569,E2 18939.569} C_VEL
LIN {X 0,Y 429.036,Z 959.35,A -85,B 0,C 180,E1 18941.938,E2 18941.938} C_VEL
LIN {X 0,Y 417.21,Z 999.907,A -85,B 0,C 180,E1 18945.148,E2 18945.148} C_VEL
LIN {X 0,Y 404.147,Z 1038.082,A -85,B 0,C 180,E1 18949.351,E2 18949.351} C_VEL
LIN {X 0,Y 391.514,Z 1071.969,A -85,B 0,C 180,E1 18954.512,E2 18954.512} C_VEL
LIN {X 0,Y 381.095,Z 1100.477,A -85,B 0,C 180,E1 18960.527,E2 18960.527} C_VEL
LIN {X 0,Y 373.279,Z 1123.54,A -85,B 0,C 180,E1 18967.316,E2 18967.316} C_VEL
LIN {X 0,Y 368.968,Z 1140.09,A -85,B 0,C 180,E1 18974.455,E2 18974.455} C_VEL
LIN {X 0,Y 367.528,Z 1149.007,A -85,B 0,C 180,E1 18980.506,E2 18980.506} C_VEL
LIN {X 0,Y 367.146,Z 1153.028,A -85,B 0,C 180,E1 18985.264,E2 18985.264} C_VEL
LIN {X 0,Y 367.325,Z 1154.405,A -85,B 0,C 180,E1 18989.998,E2 18989.998} C_VEL
LIN {X 0,Y 367.159,Z 1153.037,A -85,B 0,C 180,E1 18994.732,E2 18994.732} C_VEL
LIN {X 0,Y 367.688,Z 1147.634,A -85,B 0,C 180,E1 19000.684,E2 19000.684} C_VEL
LIN {X 0,Y 369.731,Z 1136.684,A -85,B 0,C 180,E1 19007.282,E2 19007.282} C_VEL
LIN {X 0,Y 374.369,Z 1120.024,A -85,B 0,C 180,E1 19013.872,E2 19013.872} C_VEL
LIN {X 0,Y 381.742,Z 1098.464,A -85,B 0,C 180,E1 19019.972,E2 19019.972} C_VEL
LIN {X 0,Y 392.08,Z 1070.43,A -85,B 0,C 180,E1 19025.776,E2 19025.776} C_VEL
LIN {X 0,Y 404.505,Z 1037.216,A -85,B 0,C 180,E1 19030.778,E2 19030.778} C_VEL
LIN {X 0,Y 417.667,Z 998.713,A -85,B 0,C 180,E1 19034.979,E2 19034.979} C_VEL
LIN {X 0,Y 430.067,Z 956.105,A -85,B 0,C 180,E1 19038.281,E2 19038.281} C_VEL
LIN {X 0,Y 434.92,Z 936.26,A -85,B 0,C 180,E1 19039.449,E2 19039.449} C_VEL
LIN {X 0,Y 435.394,Z 925.005,A -85,B 0,C 180,E1 19040.346,E2 19040.346} C_VEL
LIN {X 0,Y 431.056,Z 908.486,A -85,B 0,C 180,E1 19042.307,E2 19042.307} C_VEL
LIN {X 0,Y 419.818,Z 878.926,A -85,B 0,C 180,E1 19046.325,E2 19046.325} C_VEL
LIN {X 0,Y 405.898,Z 851.788,A -85,B 0,C 180,E1 19050.822,E2 19050.822} C_VEL
LIN {X 0,Y 392.321,Z 830.244,A -85,B 0,C 180,E1 19055.406,E2 19055.406} C_VEL
LIN {X 0,Y 379.922,Z 812.401,A -85,B 0,C 180,E1 19060.423,E2 19060.423} C_VEL
LIN {X 0,Y 374.221,Z 805.096,A -85,B 0,C 180,E1 19063.244,E2 19063.244} C_VEL
LIN {X 0,Y 370.211,Z 798.916,A -85,B 0,C 180,E1 19065.644,E2 19065.644} C_VEL
LIN {X 0,Y 365.184,Z 793.389,A -85,B 0,C 180,E1 19069.174,E2 19069.174} C_VEL
LIN {X 0,Y 364.213,Z 790.921,A -85,B 0,C 180,E1 19070.129,E2 19070.129} C_VEL
LIN {X 0,Y 359.219,Z 785.774,A -85,B 0,C 180,E1 19076.079,E2 19076.079} C_VEL
LIN {X 0,Y 358.964,Z 783.31,A -85,B 0,C 180,E1 19077.59,E2 19077.59} C_VEL
LIN {X 0,Y 359.004,Z 783.31,A -85,B 0,C 180,E1 19082.428,E2 19082.428} C_VEL
LIN {X 0,Y 358.737,Z 784.116,A -85,B 0,C 180,E1 19085.755,E2 19085.755} C_VEL
LIN {X 0,Y 361.803,Z 789.857,A -85,B 0,C 180,E1 19090.871,E2 19090.871} C_VEL
LIN {X 0,Y 364.666,Z 791.959,A -85,B 0,C 180,E1 19093.52,E2 19093.52} C_VEL
LIN {X 0,Y 367.505,Z 797.134,A -85,B 0,C 180,E1 19095.859,E2 19095.859} C_VEL
LIN {X 0,Y 370.341,Z 799.715,A -85,B 0,C 180,E1 19097.675,E2 19097.675} C_VEL
LIN {X 0,Y 374.663,Z 805.482,A -85,B 0,C 180,E1 19100.162,E2 19100.162} C_VEL
LIN {X 0,Y 385.368,Z 820.141,A -85,B 0,C 180,E1 19105.101,E2 19105.101} C_VEL
LIN {X 0,Y 400.217,Z 842.098,A -85,B 0,C 180,E1 19110.428,E2 19110.428} C_VEL
LIN {X 0,Y 414.497,Z 866.676,A -85,B 0,C 180,E1 19114.928,E2 19114.928} C_VEL
LIN {X 0,Y 427.269,Z 895.343,A -85,B 0,C 180,E1 19119.123,E2 19119.123} C_VEL
LIN {X 0,Y 434.086,Z 917.594,A -85,B 0,C 180,E1 19121.89,E2 19121.89} C_VEL
LIN {X 0,Y 424.264,Z 957.155,A -85,B 0,C 180,E1 19124.08,E2 19124.08} C_VEL
LIN {X 0,Y 412.515,Z 994.681,A -85,B 0,C 180,E1 19127.061,E2 19127.061} C_VEL
LIN {X 0,Y 399.786,Z 1029.188,A -85,B 0,C 180,E1 19130.9,E2 19130.9} C_VEL
LIN {X 0,Y 386.997,Z 1060.376,A -85,B 0,C 180,E1 19135.733,E2 19135.733} C_VEL
LIN {X 0,Y 375.272,Z 1087.638,A -85,B 0,C 180,E1 19141.682,E2 19141.682} C_VEL
LIN {X 0,Y 366.972,Z 1108.375,A -85,B 0,C 180,E1 19148.188,E2 19148.188} C_VEL
LIN {X 0,Y 362.159,Z 1122.479,A -85,B 0,C 180,E1 19154.733,E2 19154.733} C_VEL
LIN {X 0,Y 360.011,Z 1131.017,A -85,B 0,C 180,E1 19161.133,E2 19161.133} C_VEL
LIN {X 0,Y 359.389,Z 1135.035,A -85,B 0,C 180,E1 19167.586,E2 19167.586} C_VEL
LIN {X 0,Y 359.459,Z 1135.013,A -85,B 0,C 180,E1 19172.418,E2 19172.418} C_VEL
LIN {X 0,Y 360.063,Z 1130.899,A -85,B 0,C 180,E1 19178.879,E2 19178.879} C_VEL
LIN {X 0,Y 362.209,Z 1122.211,A -85,B 0,C 180,E1 19185.306,E2 19185.306} C_VEL
LIN {X 0,Y 367.015,Z 1108.106,A -85,B 0,C 180,E1 19191.813,E2 19191.813} C_VEL
LIN {X 0,Y 375.433,Z 1087.265,A -85,B 0,C 180,E1 19198.309,E2 19198.309} C_VEL
LIN {X 0,Y 386.695,Z 1060.858,A -85,B 0,C 180,E1 19204.073,E2 19204.073} C_VEL
LIN {X 0,Y 399.714,Z 1029.185,A -85,B 0,C 180,E1 19208.993,E2 19208.993} C_VEL
LIN {X 0,Y 412.661,Z 994.111,A -85,B 0,C 180,E1 19212.882,E2 19212.882} C_VEL
LIN {X 0,Y 424.655,Z 955.451,A -85,B 0,C 180,E1 19215.931,E2 19215.931} C_VEL
LIN {X 0,Y 434.148,Z 916.384,A -85,B 0,C 180,E1 19218.074,E2 19218.074} C_VEL
LIN {X 0,Y 423.325,Z 885.736,A -85,B 0,C 180,E1 19222.07,E2 19222.07} C_VEL
LIN {X 0,Y 408.993,Z 856.607,A -85,B 0,C 180,E1 19226.634,E2 19226.634} C_VEL
LIN {X 0,Y 393.297,Z 831.559,A -85,B 0,C 180,E1 19231.756,E2 19231.756} C_VEL
LIN {X 0,Y 379.643,Z 812.285,A -85,B 0,C 180,E1 19237.17,E2 19237.17} C_VEL
LIN {X 0,Y 374.039,Z 805.048,A -85,B 0,C 180,E1 19239.926,E2 19239.926} C_VEL
LIN {X 0,Y 370.092,Z 798.997,A -85,B 0,C 180,E1 19242.264,E2 19242.264} C_VEL
LIN {X 0,Y 364.939,Z 793.351,A -85,B 0,C 180,E1 19245.851,E2 19245.851} C_VEL
LIN {X 0,Y 364.12,Z 790.963,A -85,B 0,C 180,E1 19246.669,E2 19246.669} C_VEL
LIN {X 0,Y 359.041,Z 785.947,A -85,B 0,C 180,E1 19252.49,E2 19252.49} C_VEL
LIN {X 0,Y 358.693,Z 783.31,A -85,B 0,C 180,E1 19254.036,E2 19254.036} C_VEL
LIN {X 0,Y 359.233,Z 783.31,A -85,B 0,C 180,E1 19259.991,E2 19259.991} C_VEL
LIN {X 0,Y 358.919,Z 784.061,A -85,B 0,C 180,E1 19263.621,E2 19263.621} C_VEL
LIN {X 0,Y 361.657,Z 789.613,A -85,B 0,C 180,E1 19267.816,E2 19267.816} C_VEL
LIN {X 0,Y 364.776,Z 791.919,A -85,B 0,C 180,E1 19270.611,E2 19270.611} C_VEL
LIN {X 0,Y 368.103,Z 797.419,A -85,B 0,C 180,E1 19273.226,E2 19273.226} C_VEL
LIN {X 0,Y 370.502,Z 799.767,A -85,B 0,C 180,E1 19274.723,E2 19274.723} C_VEL
LIN {X 0,Y 374.826,Z 805.449,A -85,B 0,C 180,E1 19277.182,E2 19277.182} C_VEL
LIN {X 0,Y 385.781,Z 820.804,A -85,B 0,C 180,E1 19282.2,E2 19282.2} C_VEL
LIN {X 0,Y 399.739,Z 841.563,A -85,B 0,C 180,E1 19287.232,E2 19287.232} C_VEL
LIN {X 0,Y 414.082,Z 867.095,A -85,B 0,C 180,E1 19291.869,E2 19291.869} C_VEL
LIN {X 0,Y 426.987,Z 896.931,A -85,B 0,C 180,E1 19296.204,E2 19296.204} C_VEL
LIN {X 0,Y 433.354,Z 919.269,A -85,B 0,C 180,E1 19298.925,E2 19298.925} C_VEL
LIN {X 0,Y 423.197,Z 960.651,A -85,B 0,C 180,E1 19301.246,E2 19301.246} C_VEL
LIN {X 0,Y 410.933,Z 1001.235,A -85,B 0,C 180,E1 19304.515,E2 19304.515} C_VEL
LIN {X 0,Y 397.967,Z 1037.881,A -85,B 0,C 180,E1 19308.599,E2 19308.599} C_VEL
LIN {X 0,Y 384.906,Z 1071.709,A -85,B 0,C 180,E1 19313.807,E2 19313.807} C_VEL
